(* IEC 61131-3 sources: TIA2AX/tests/V18/test_projects/expected/HW_2200330/ST70_PLC, 7 files *)

(* ---- HwIdentifiers.st ---- *)
TYPE
	HwIdentifiers : WORD
	(
		ST70_PLC_Profilschiene_0 :=	WORD#256,
		ST70_PLC :=	WORD#48,
		ST70_PLC_Card_reader_writer_1 :=	WORD#51,
		ST70_PLC_CPU_display_1 :=	WORD#54,
		ST70_PLC_OPC_UA_1 :=	WORD#117,
		ST70_PLC_DP_interface_1 :=	WORD#60,
		ST70_PLC_PROFINET_interface_1 :=	WORD#64,
		ST70_PLC_PROFINET_interface_1_Port_1 :=	WORD#65,
		ST70_PLC_PROFINET_interface_1_Port_2 :=	WORD#66,
		ST70_PLC_PROFINET_interface_2 :=	WORD#72,
		ST70_PLC_PROFINET_interface_2_Port_1 :=	WORD#73,
		ST70_Switch_SCALANCE_X_rack :=	WORD#406,
		ST70_Switch :=	WORD#407,
		ST70_Switch_ST70_Switch :=	WORD#408,
		ST70_Switch_SCALANCE_interface_1 :=	WORD#409,
		ST70_Switch_SCALANCE_interface_1_Port_1 :=	WORD#410,
		ST70_Switch_SCALANCE_interface_1_Port_2 :=	WORD#411,
		ST70_Switch_SCALANCE_interface_1_Port_3 :=	WORD#412,
		ST70_Switch_SCALANCE_interface_1_Port_4 :=	WORD#413,
		ST70_Switch_SCALANCE_interface_1_Port_5 :=	WORD#414,
		ST70_Switch_SCALANCE_interface_1_Port_6 :=	WORD#415,
		ST70_Switch_SCALANCE_interface_1_Port_7 :=	WORD#416,
		ST70_Switch_SCALANCE_interface_1_Port_8 :=	WORD#417,
		ST70_Switch_SCALANCE_interface_1_Port_9 :=	WORD#418,
		ST70_Switch_SCALANCE_interface_1_Port_10 :=	WORD#419,
		ST70_Switch_SCALANCE_interface_1_Port_11 :=	WORD#420,
		ST70_Switch_SCALANCE_interface_1_Port_12 :=	WORD#421,
		ST70_Switch_SCALANCE_interface_1_Port_13 :=	WORD#422,
		ST70_Switch_SCALANCE_interface_1_Port_14 :=	WORD#423,
		ST70_Switch_SCALANCE_interface_1_Port_15 :=	WORD#424,
		ST70_Switch_SCALANCE_interface_1_Port_16 :=	WORD#425,
		ST70_HMI_ConnectionBox_Connection_Box :=	WORD#265,
		ST70_HMI_ConnectionBox :=	WORD#258,
		ST70_HMI_ConnectionBox_ST70_HMI_ConnectionBox :=	WORD#259,
		ST70_HMI_ConnectionBox_SCALANCE_interface_1 :=	WORD#260,
		ST70_HMI_ConnectionBox_SCALANCE_interface_1_Port_1 :=	WORD#261,
		ST70_HMI_ConnectionBox_SCALANCE_interface_1_Port_2 :=	WORD#262,
		ST70_HMI_ConnectionBox_SCALANCE_interface_1_Port_3 :=	WORD#263,
		ST70_ET200SP_Rack_0 :=	WORD#272,
		ST70_ET200SP :=	WORD#273,
		ST70_ET200SP_ST70_ET200SP :=	WORD#274,
		ST70_ET200SP_PROFINET_interface :=	WORD#275,
		ST70_ET200SP_PROFINET_interface_Port_1 :=	WORD#277,
		ST70_ET200SP_PROFINET_interface_Port_2 :=	WORD#276,
		ST70_ET200SP_BA_2xRJ45 :=	WORD#277,
		ST70_ET200SP_CM_4xIO_Link_1 :=	WORD#278,
		ST70_ET200SP_DI_16x24VDC_ST_1 :=	WORD#279,
		ST70_ET200SP_DI_16x24VDC_ST_2 :=	WORD#280,
		ST70_ET200SP_DI_8x24VDC_ST_3 :=	WORD#281,
		ST70_ET200SP_DI_16x24VDC_ST_4 :=	WORD#266,
		ST70_ET200SP_DQ_16x24VDC_0_5A_ST_1 :=	WORD#267,
		ST70_ET200SP_DQ_16x24VDC_0_5A_ST_2 :=	WORD#268,
		ST70_ET200SP_DQ_16x24VDC_0_5A_ST_3 :=	WORD#269,
		ST70_ET200SP_Servermodul_1 :=	WORD#270,
		ST70_CPX_PN_IO_Interface :=	WORD#285,
		ST70_CPX_PN_IO_Interface_Port_1 :=	WORD#286,
		ST70_CPX_PN_IO_Interface_Port_2 :=	WORD#287,
		ST70_CPX_CPX :=	WORD#288,
		ST70_CPX_MPA1S_VMPA1_FB_EMS_8_8DO_1 :=	WORD#289,
		ST70_CPX_MPA1S_VMPA1_FB_EMS_8_8DO_2 :=	WORD#290,
		ST70_CPX_MPA1S_VMPA1_FB_EMS_8_8DO_3 :=	WORD#291,
		ST70_CPX_MPA2S_VMPA2_FB_EMS_4_4DO_1 :=	WORD#292,
		ST70_CPX_MPA1G_VMPA1_FB_EMG_8_8DO_3 :=	WORD#293,
		ST70_1_DM260_PB_Rack :=	WORD#295,
		ST70_1_DM260_PB :=	WORD#296,
		ST70_1_DM260_PB_Interface :=	WORD#297,
		ST70_1_DM260_PB_Interface_Port_1 :=	WORD#298,
		ST70_1_DM260_PB_DataMan_260 :=	WORD#299,
		ST70_1_DM260_PB_Acquisition_Control_1 :=	WORD#300,
		ST70_1_DM260_PB_Acquisition_Status_1 :=	WORD#301,
		ST70_1_DM260_PB_Results_Control_1 :=	WORD#302,
		ST70_1_DM260_PB_Results_Status_1 :=	WORD#303,
		ST70_1_DM260_PB_Soft_Event_Control_1 :=	WORD#304,
		ST70_1_DM260_PB_User_Data_64_bytes_1 :=	WORD#305,
		ST70_1_DM260_PB_Result_Data_64_bytes_1 :=	WORD#306,
		ST70_2_DM260_PB_Rack :=	WORD#308,
		ST70_2_DM260_PB :=	WORD#309,
		ST70_2_DM260_PB_Interface :=	WORD#310,
		ST70_2_DM260_PB_Interface_Port_1 :=	WORD#311,
		ST70_2_DM260_PB_DataMan_260 :=	WORD#312,
		ST70_2_DM260_PB_Acquisition_Control_1 :=	WORD#313,
		ST70_2_DM260_PB_Acquisition_Status_1 :=	WORD#314,
		ST70_2_DM260_PB_Results_Control_1 :=	WORD#315,
		ST70_2_DM260_PB_Results_Status_1 :=	WORD#316,
		ST70_2_DM260_PB_Soft_Event_Control_1 :=	WORD#317,
		ST70_2_DM260_PB_User_Data_64_bytes_1 :=	WORD#318,
		ST70_2_DM260_PB_Result_Data_64_bytes_1 :=	WORD#319,
		ST70_1_CMMT_3GF1_PN_IO_Interface :=	WORD#323,
		ST70_1_CMMT_3GF1_PN_IO_Interface_Port_1 :=	WORD#324,
		ST70_1_CMMT_3GF1_PN_IO_Interface_Port_2 :=	WORD#325,
		ST70_1_CMMT_3GF1_CMMT_AS_V1 :=	WORD#326,
		ST70_1_CMMT_3GF1_DO_SERVO_1_Module_Access_Point :=	WORD#328,
		ST70_1_CMMT_3GF1_DO_SERVO_1_Siemens_telegram_111_PZD_12_12 :=	WORD#329,
		ST70_1_CMMT_3GF1_Siemens_telegram_111_PZD_12_12 :=	WORD#329,
		ST70_1_CMMT_3GF2_PN_IO_Interface :=	WORD#333,
		ST70_1_CMMT_3GF2_PN_IO_Interface_Port_1 :=	WORD#334,
		ST70_1_CMMT_3GF2_PN_IO_Interface_Port_2 :=	WORD#335,
		ST70_1_CMMT_3GF2_CMMT_AS_V1 :=	WORD#336,
		ST70_1_CMMT_3GF2_DO_SERVO_1_Module_Access_Point :=	WORD#338,
		ST70_1_CMMT_3GF2_DO_SERVO_1_Siemens_telegram_111_PZD_12_12 :=	WORD#339,
		ST70_1_CMMT_3GF2_Siemens_telegram_111_PZD_12_12 :=	WORD#339,
		ST70_3_DM260_PB_Rack :=	WORD#341,
		ST70_3_DM260_PB :=	WORD#342,
		ST70_3_DM260_PB_Interface :=	WORD#343,
		ST70_3_DM260_PB_Interface_Port_1 :=	WORD#344,
		ST70_3_DM260_PB_DataMan_260 :=	WORD#345,
		ST70_3_DM260_PB_Acquisition_Control_1 :=	WORD#346,
		ST70_3_DM260_PB_Acquisition_Status_1 :=	WORD#347,
		ST70_3_DM260_PB_Results_Control_1 :=	WORD#348,
		ST70_3_DM260_PB_Results_Status_1 :=	WORD#349,
		ST70_3_DM260_PB_Soft_Event_Control_1 :=	WORD#350,
		ST70_3_DM260_PB_User_Data_64_bytes_1 :=	WORD#351,
		ST70_3_DM260_PB_Result_Data_64_bytes_1 :=	WORD#352,
		ST70_1_DM260_EB_Rack :=	WORD#354,
		ST70_1_DM260_EB :=	WORD#355,
		ST70_1_DM260_EB_Interface :=	WORD#356,
		ST70_1_DM260_EB_Interface_Port_1 :=	WORD#357,
		ST70_1_DM260_EB_DataMan_260 :=	WORD#358,
		ST70_1_DM260_EB_Acquisition_Control_1 :=	WORD#359,
		ST70_1_DM260_EB_Acquisition_Status_1 :=	WORD#360,
		ST70_1_DM260_EB_Results_Control_1 :=	WORD#361,
		ST70_1_DM260_EB_Results_Status_1 :=	WORD#362,
		ST70_1_DM260_EB_Soft_Event_Control_1 :=	WORD#363,
		ST70_1_DM260_EB_User_Data_64_bytes_1 :=	WORD#364,
		ST70_1_DM260_EB_Result_Data_64_bytes_1 :=	WORD#365,
		ST70_2_DM260_EB_Rack :=	WORD#367,
		ST70_2_DM260_EB :=	WORD#368,
		ST70_2_DM260_EB_Interface :=	WORD#369,
		ST70_2_DM260_EB_Interface_Port_1 :=	WORD#370,
		ST70_2_DM260_EB_DataMan_260 :=	WORD#371,
		ST70_2_DM260_EB_Acquisition_Control_1 :=	WORD#372,
		ST70_2_DM260_EB_Acquisition_Status_1 :=	WORD#373,
		ST70_2_DM260_EB_Results_Control_1 :=	WORD#374,
		ST70_2_DM260_EB_Results_Status_1 :=	WORD#375,
		ST70_2_DM260_EB_Soft_Event_Control_1 :=	WORD#376,
		ST70_2_DM260_EB_User_Data_64_bytes_1 :=	WORD#377,
		ST70_2_DM260_EB_Result_Data_64_bytes_1 :=	WORD#378,
		ST70_3_DM260_EB_Rack :=	WORD#380,
		ST70_3_DM260_EB :=	WORD#381,
		ST70_3_DM260_EB_Interface :=	WORD#382,
		ST70_3_DM260_EB_Interface_Port_1 :=	WORD#383,
		ST70_3_DM260_EB_DataMan_260 :=	WORD#384,
		ST70_3_DM260_EB_Acquisition_Control_1 :=	WORD#385,
		ST70_3_DM260_EB_Acquisition_Status_1 :=	WORD#386,
		ST70_3_DM260_EB_Results_Control_1 :=	WORD#387,
		ST70_3_DM260_EB_Results_Status_1 :=	WORD#388,
		ST70_3_DM260_EB_Soft_Event_Control_1 :=	WORD#389,
		ST70_3_DM260_EB_User_Data_64_bytes_1 :=	WORD#390,
		ST70_3_DM260_EB_Result_Data_64_bytes_1 :=	WORD#391,
		ST70_1_CMMT_3GF3_PN_IO_Interface :=	WORD#395,
		ST70_1_CMMT_3GF3_PN_IO_Interface_Port_1 :=	WORD#396,
		ST70_1_CMMT_3GF3_PN_IO_Interface_Port_2 :=	WORD#397,
		ST70_1_CMMT_3GF3_CMMT_AS_V1 :=	WORD#398,
		ST70_1_CMMT_3GF3_DO_SERVO_1_Module_Access_Point :=	WORD#400,
		ST70_1_CMMT_3GF3_DO_SERVO_1_Siemens_telegram_111_PZD_12_12 :=	WORD#401,
		ST70_1_CMMT_3GF3_Siemens_telegram_111_PZD_12_12 :=	WORD#401,
		NONE:= WORD#0
	);
END_TYPE

(* ---- HwInputs.st ---- *)
TYPE
	HwInputs : STRUCT
		ST70_ET200SP_CM_4xIO_Link_1 AT %B100 : ARRAY[0..31] OF BYTE;
		ST70_ET200SP_DI_16x24VDC_ST_1 AT %B0 : WORD;
		ST70_ET200SP_DI_16x24VDC_ST_2 AT %B2 : WORD;
		ST70_ET200SP_DI_8x24VDC_ST_3 AT %B4 : BYTE;
		ST70_ET200SP_DI_16x24VDC_ST_4 AT %B5 : WORD;
		ST70_1_DM260_PB_Acquisition_Status_1 AT %B1000 : ARRAY[0..2] OF BYTE;
		ST70_1_DM260_PB_Results_Status_1 AT %B1003 : BYTE;
		ST70_1_DM260_PB_Soft_Event_Control_1 AT %B1004 : BYTE;
		ST70_1_DM260_PB_Result_Data_64_bytes_1 AT %B1010 : ARRAY[0..71] OF BYTE;
		ST70_2_DM260_PB_Acquisition_Status_1 AT %B2000 : ARRAY[0..2] OF BYTE;
		ST70_2_DM260_PB_Results_Status_1 AT %B2003 : BYTE;
		ST70_2_DM260_PB_Soft_Event_Control_1 AT %B2004 : BYTE;
		ST70_2_DM260_PB_Result_Data_64_bytes_1 AT %B2010 : ARRAY[0..71] OF BYTE;
		ST70_1_CMMT_3GF1_DO_SERVO_1_Siemens_telegram_111_PZD_12_12 AT %B1500 : ARRAY[0..23] OF BYTE;
		ST70_1_CMMT_3GF2_DO_SERVO_1_Siemens_telegram_111_PZD_12_12 AT %B1600 : ARRAY[0..23] OF BYTE;
		ST70_3_DM260_PB_Acquisition_Status_1 AT %B3000 : ARRAY[0..2] OF BYTE;
		ST70_3_DM260_PB_Results_Status_1 AT %B3003 : BYTE;
		ST70_3_DM260_PB_Soft_Event_Control_1 AT %B3004 : BYTE;
		ST70_3_DM260_PB_Result_Data_64_bytes_1 AT %B3010 : ARRAY[0..71] OF BYTE;
		ST70_1_DM260_EB_Acquisition_Status_1 AT %B1200 : ARRAY[0..2] OF BYTE;
		ST70_1_DM260_EB_Results_Status_1 AT %B1203 : BYTE;
		ST70_1_DM260_EB_Soft_Event_Control_1 AT %B1204 : BYTE;
		ST70_1_DM260_EB_Result_Data_64_bytes_1 AT %B1210 : ARRAY[0..71] OF BYTE;
		ST70_2_DM260_EB_Acquisition_Status_1 AT %B2200 : ARRAY[0..2] OF BYTE;
		ST70_2_DM260_EB_Results_Status_1 AT %B2203 : BYTE;
		ST70_2_DM260_EB_Soft_Event_Control_1 AT %B2204 : BYTE;
		ST70_2_DM260_EB_Result_Data_64_bytes_1 AT %B2210 : ARRAY[0..71] OF BYTE;
		ST70_3_DM260_EB_Acquisition_Status_1 AT %B3200 : ARRAY[0..2] OF BYTE;
		ST70_3_DM260_EB_Results_Status_1 AT %B3203 : BYTE;
		ST70_3_DM260_EB_Soft_Event_Control_1 AT %B3204 : BYTE;
		ST70_3_DM260_EB_Result_Data_64_bytes_1 AT %B3210 : ARRAY[0..71] OF BYTE;
		ST70_1_CMMT_3GF3_DO_SERVO_1_Siemens_telegram_111_PZD_12_12 AT %B1624 : ARRAY[0..23] OF BYTE;
	END_STRUCT;
END_TYPE

(* ---- HwOutputs.st ---- *)
TYPE
	HwOutputs : STRUCT
		ST70_ET200SP_CM_4xIO_Link_1 AT %B100 : ARRAY[0..31] OF BYTE;
		ST70_ET200SP_DQ_16x24VDC_0_5A_ST_1 AT %B0 : WORD;
		ST70_ET200SP_DQ_16x24VDC_0_5A_ST_2 AT %B2 : WORD;
		ST70_ET200SP_DQ_16x24VDC_0_5A_ST_3 AT %B4 : WORD;
		ST70_CPX_MPA1S_VMPA1_FB_EMS_8_8DO_1 AT %B200 : BYTE;
		ST70_CPX_MPA1S_VMPA1_FB_EMS_8_8DO_2 AT %B201 : BYTE;
		ST70_CPX_MPA1S_VMPA1_FB_EMS_8_8DO_3 AT %B202 : BYTE;
		ST70_CPX_MPA2S_VMPA2_FB_EMS_4_4DO_1 AT %B6 : BYTE;
		ST70_CPX_MPA1G_VMPA1_FB_EMG_8_8DO_3 AT %B204 : BYTE;
		ST70_1_DM260_PB_Acquisition_Control_1 AT %B1000 : BYTE;
		ST70_1_DM260_PB_Results_Control_1 AT %B1003 : BYTE;
		ST70_1_DM260_PB_Soft_Event_Control_1 AT %B1004 : BYTE;
		ST70_1_DM260_PB_User_Data_64_bytes_1 AT %B1010 : ARRAY[0..67] OF BYTE;
		ST70_2_DM260_PB_Acquisition_Control_1 AT %B2000 : BYTE;
		ST70_2_DM260_PB_Results_Control_1 AT %B2003 : BYTE;
		ST70_2_DM260_PB_Soft_Event_Control_1 AT %B2004 : BYTE;
		ST70_2_DM260_PB_User_Data_64_bytes_1 AT %B2010 : ARRAY[0..67] OF BYTE;
		ST70_1_CMMT_3GF1_DO_SERVO_1_Siemens_telegram_111_PZD_12_12 AT %B1500 : ARRAY[0..23] OF BYTE;
		ST70_1_CMMT_3GF2_DO_SERVO_1_Siemens_telegram_111_PZD_12_12 AT %B1600 : ARRAY[0..23] OF BYTE;
		ST70_3_DM260_PB_Acquisition_Control_1 AT %B3000 : BYTE;
		ST70_3_DM260_PB_Results_Control_1 AT %B3003 : BYTE;
		ST70_3_DM260_PB_Soft_Event_Control_1 AT %B3004 : BYTE;
		ST70_3_DM260_PB_User_Data_64_bytes_1 AT %B3010 : ARRAY[0..67] OF BYTE;
		ST70_1_DM260_EB_Acquisition_Control_1 AT %B1200 : BYTE;
		ST70_1_DM260_EB_Results_Control_1 AT %B1203 : BYTE;
		ST70_1_DM260_EB_Soft_Event_Control_1 AT %B1204 : BYTE;
		ST70_1_DM260_EB_User_Data_64_bytes_1 AT %B1210 : ARRAY[0..67] OF BYTE;
		ST70_2_DM260_EB_Acquisition_Control_1 AT %B2200 : BYTE;
		ST70_2_DM260_EB_Results_Control_1 AT %B2203 : BYTE;
		ST70_2_DM260_EB_Soft_Event_Control_1 AT %B2204 : BYTE;
		ST70_2_DM260_EB_User_Data_64_bytes_1 AT %B2210 : ARRAY[0..67] OF BYTE;
		ST70_3_DM260_EB_Acquisition_Control_1 AT %B3200 : BYTE;
		ST70_3_DM260_EB_Results_Control_1 AT %B3203 : BYTE;
		ST70_3_DM260_EB_Soft_Event_Control_1 AT %B3204 : BYTE;
		ST70_3_DM260_EB_User_Data_64_bytes_1 AT %B3210 : ARRAY[0..67] OF BYTE;
		ST70_1_CMMT_3GF3_DO_SERVO_1_Siemens_telegram_111_PZD_12_12 AT %B1624 : ARRAY[0..23] OF BYTE;
	END_STRUCT;
END_TYPE

(* ---- PlcInputs.st ---- *)
TYPE
	PlcInputs : STRUCT
		ST70_ET200SP_CM_4xIO_Link_1 : ARRAY[0..31] OF BYTE;
		ST70_ET200SP_DI_16x24VDC_ST_1 : WORD;
		ST70_ET200SP_DI_16x24VDC_ST_2 : WORD;
		ST70_ET200SP_DI_8x24VDC_ST_3 : BYTE;
		ST70_ET200SP_DI_16x24VDC_ST_4 : WORD;
		ST70_1_DM260_PB_Acquisition_Status_1 : ARRAY[0..2] OF BYTE;
		ST70_1_DM260_PB_Results_Status_1 : BYTE;
		ST70_1_DM260_PB_Soft_Event_Control_1 : BYTE;
		ST70_1_DM260_PB_Result_Data_64_bytes_1 : ARRAY[0..71] OF BYTE;
		ST70_2_DM260_PB_Acquisition_Status_1 : ARRAY[0..2] OF BYTE;
		ST70_2_DM260_PB_Results_Status_1 : BYTE;
		ST70_2_DM260_PB_Soft_Event_Control_1 : BYTE;
		ST70_2_DM260_PB_Result_Data_64_bytes_1 : ARRAY[0..71] OF BYTE;
		ST70_1_CMMT_3GF1_DO_SERVO_1_Siemens_telegram_111_PZD_12_12 : ARRAY[0..23] OF BYTE;
		ST70_1_CMMT_3GF2_DO_SERVO_1_Siemens_telegram_111_PZD_12_12 : ARRAY[0..23] OF BYTE;
		ST70_3_DM260_PB_Acquisition_Status_1 : ARRAY[0..2] OF BYTE;
		ST70_3_DM260_PB_Results_Status_1 : BYTE;
		ST70_3_DM260_PB_Soft_Event_Control_1 : BYTE;
		ST70_3_DM260_PB_Result_Data_64_bytes_1 : ARRAY[0..71] OF BYTE;
		ST70_1_DM260_EB_Acquisition_Status_1 : ARRAY[0..2] OF BYTE;
		ST70_1_DM260_EB_Results_Status_1 : BYTE;
		ST70_1_DM260_EB_Soft_Event_Control_1 : BYTE;
		ST70_1_DM260_EB_Result_Data_64_bytes_1 : ARRAY[0..71] OF BYTE;
		ST70_2_DM260_EB_Acquisition_Status_1 : ARRAY[0..2] OF BYTE;
		ST70_2_DM260_EB_Results_Status_1 : BYTE;
		ST70_2_DM260_EB_Soft_Event_Control_1 : BYTE;
		ST70_2_DM260_EB_Result_Data_64_bytes_1 : ARRAY[0..71] OF BYTE;
		ST70_3_DM260_EB_Acquisition_Status_1 : ARRAY[0..2] OF BYTE;
		ST70_3_DM260_EB_Results_Status_1 : BYTE;
		ST70_3_DM260_EB_Soft_Event_Control_1 : BYTE;
		ST70_3_DM260_EB_Result_Data_64_bytes_1 : ARRAY[0..71] OF BYTE;
		ST70_1_CMMT_3GF3_DO_SERVO_1_Siemens_telegram_111_PZD_12_12 : ARRAY[0..23] OF BYTE;
	END_STRUCT;
END_TYPE

(* ---- PlcOutputs.st ---- *)
TYPE
	PlcOutputs : STRUCT
		ST70_ET200SP_CM_4xIO_Link_1 : ARRAY[0..31] OF BYTE;
		ST70_ET200SP_DQ_16x24VDC_0_5A_ST_1 : WORD;
		ST70_ET200SP_DQ_16x24VDC_0_5A_ST_2 : WORD;
		ST70_ET200SP_DQ_16x24VDC_0_5A_ST_3 : WORD;
		ST70_CPX_MPA1S_VMPA1_FB_EMS_8_8DO_1 : BYTE;
		ST70_CPX_MPA1S_VMPA1_FB_EMS_8_8DO_2 : BYTE;
		ST70_CPX_MPA1S_VMPA1_FB_EMS_8_8DO_3 : BYTE;
		ST70_CPX_MPA2S_VMPA2_FB_EMS_4_4DO_1 : BYTE;
		ST70_CPX_MPA1G_VMPA1_FB_EMG_8_8DO_3 : BYTE;
		ST70_1_DM260_PB_Acquisition_Control_1 : BYTE;
		ST70_1_DM260_PB_Results_Control_1 : BYTE;
		ST70_1_DM260_PB_Soft_Event_Control_1 : BYTE;
		ST70_1_DM260_PB_User_Data_64_bytes_1 : ARRAY[0..67] OF BYTE;
		ST70_2_DM260_PB_Acquisition_Control_1 : BYTE;
		ST70_2_DM260_PB_Results_Control_1 : BYTE;
		ST70_2_DM260_PB_Soft_Event_Control_1 : BYTE;
		ST70_2_DM260_PB_User_Data_64_bytes_1 : ARRAY[0..67] OF BYTE;
		ST70_1_CMMT_3GF1_DO_SERVO_1_Siemens_telegram_111_PZD_12_12 : ARRAY[0..23] OF BYTE;
		ST70_1_CMMT_3GF2_DO_SERVO_1_Siemens_telegram_111_PZD_12_12 : ARRAY[0..23] OF BYTE;
		ST70_3_DM260_PB_Acquisition_Control_1 : BYTE;
		ST70_3_DM260_PB_Results_Control_1 : BYTE;
		ST70_3_DM260_PB_Soft_Event_Control_1 : BYTE;
		ST70_3_DM260_PB_User_Data_64_bytes_1 : ARRAY[0..67] OF BYTE;
		ST70_1_DM260_EB_Acquisition_Control_1 : BYTE;
		ST70_1_DM260_EB_Results_Control_1 : BYTE;
		ST70_1_DM260_EB_Soft_Event_Control_1 : BYTE;
		ST70_1_DM260_EB_User_Data_64_bytes_1 : ARRAY[0..67] OF BYTE;
		ST70_2_DM260_EB_Acquisition_Control_1 : BYTE;
		ST70_2_DM260_EB_Results_Control_1 : BYTE;
		ST70_2_DM260_EB_Soft_Event_Control_1 : BYTE;
		ST70_2_DM260_EB_User_Data_64_bytes_1 : ARRAY[0..67] OF BYTE;
		ST70_3_DM260_EB_Acquisition_Control_1 : BYTE;
		ST70_3_DM260_EB_Results_Control_1 : BYTE;
		ST70_3_DM260_EB_Soft_Event_Control_1 : BYTE;
		ST70_3_DM260_EB_User_Data_64_bytes_1 : ARRAY[0..67] OF BYTE;
		ST70_1_CMMT_3GF3_DO_SERVO_1_Siemens_telegram_111_PZD_12_12 : ARRAY[0..23] OF BYTE;
	END_STRUCT;
END_TYPE

(* ---- CopyInputs.st ---- *)
FUNCTION CopyInputs
	VAR_EXTERNAL
		HwInputs : HwInputs;
		PlcInputs : PlcInputs;
	END_VAR
	PlcInputs.ST70_ET200SP_CM_4xIO_Link_1[0] := HwInputs.ST70_ET200SP_CM_4xIO_Link_1[0];
	PlcInputs.ST70_ET200SP_CM_4xIO_Link_1[1] := HwInputs.ST70_ET200SP_CM_4xIO_Link_1[1];
	PlcInputs.ST70_ET200SP_CM_4xIO_Link_1[2] := HwInputs.ST70_ET200SP_CM_4xIO_Link_1[2];
	PlcInputs.ST70_ET200SP_CM_4xIO_Link_1[3] := HwInputs.ST70_ET200SP_CM_4xIO_Link_1[3];
	PlcInputs.ST70_ET200SP_CM_4xIO_Link_1[4] := HwInputs.ST70_ET200SP_CM_4xIO_Link_1[4];
	PlcInputs.ST70_ET200SP_CM_4xIO_Link_1[5] := HwInputs.ST70_ET200SP_CM_4xIO_Link_1[5];
	PlcInputs.ST70_ET200SP_CM_4xIO_Link_1[6] := HwInputs.ST70_ET200SP_CM_4xIO_Link_1[6];
	PlcInputs.ST70_ET200SP_CM_4xIO_Link_1[7] := HwInputs.ST70_ET200SP_CM_4xIO_Link_1[7];
	PlcInputs.ST70_ET200SP_CM_4xIO_Link_1[8] := HwInputs.ST70_ET200SP_CM_4xIO_Link_1[8];
	PlcInputs.ST70_ET200SP_CM_4xIO_Link_1[9] := HwInputs.ST70_ET200SP_CM_4xIO_Link_1[9];
	PlcInputs.ST70_ET200SP_CM_4xIO_Link_1[10] := HwInputs.ST70_ET200SP_CM_4xIO_Link_1[10];
	PlcInputs.ST70_ET200SP_CM_4xIO_Link_1[11] := HwInputs.ST70_ET200SP_CM_4xIO_Link_1[11];
	PlcInputs.ST70_ET200SP_CM_4xIO_Link_1[12] := HwInputs.ST70_ET200SP_CM_4xIO_Link_1[12];
	PlcInputs.ST70_ET200SP_CM_4xIO_Link_1[13] := HwInputs.ST70_ET200SP_CM_4xIO_Link_1[13];
	PlcInputs.ST70_ET200SP_CM_4xIO_Link_1[14] := HwInputs.ST70_ET200SP_CM_4xIO_Link_1[14];
	PlcInputs.ST70_ET200SP_CM_4xIO_Link_1[15] := HwInputs.ST70_ET200SP_CM_4xIO_Link_1[15];
	PlcInputs.ST70_ET200SP_CM_4xIO_Link_1[16] := HwInputs.ST70_ET200SP_CM_4xIO_Link_1[16];
	PlcInputs.ST70_ET200SP_CM_4xIO_Link_1[17] := HwInputs.ST70_ET200SP_CM_4xIO_Link_1[17];
	PlcInputs.ST70_ET200SP_CM_4xIO_Link_1[18] := HwInputs.ST70_ET200SP_CM_4xIO_Link_1[18];
	PlcInputs.ST70_ET200SP_CM_4xIO_Link_1[19] := HwInputs.ST70_ET200SP_CM_4xIO_Link_1[19];
	PlcInputs.ST70_ET200SP_CM_4xIO_Link_1[20] := HwInputs.ST70_ET200SP_CM_4xIO_Link_1[20];
	PlcInputs.ST70_ET200SP_CM_4xIO_Link_1[21] := HwInputs.ST70_ET200SP_CM_4xIO_Link_1[21];
	PlcInputs.ST70_ET200SP_CM_4xIO_Link_1[22] := HwInputs.ST70_ET200SP_CM_4xIO_Link_1[22];
	PlcInputs.ST70_ET200SP_CM_4xIO_Link_1[23] := HwInputs.ST70_ET200SP_CM_4xIO_Link_1[23];
	PlcInputs.ST70_ET200SP_CM_4xIO_Link_1[24] := HwInputs.ST70_ET200SP_CM_4xIO_Link_1[24];
	PlcInputs.ST70_ET200SP_CM_4xIO_Link_1[25] := HwInputs.ST70_ET200SP_CM_4xIO_Link_1[25];
	PlcInputs.ST70_ET200SP_CM_4xIO_Link_1[26] := HwInputs.ST70_ET200SP_CM_4xIO_Link_1[26];
	PlcInputs.ST70_ET200SP_CM_4xIO_Link_1[27] := HwInputs.ST70_ET200SP_CM_4xIO_Link_1[27];
	PlcInputs.ST70_ET200SP_CM_4xIO_Link_1[28] := HwInputs.ST70_ET200SP_CM_4xIO_Link_1[28];
	PlcInputs.ST70_ET200SP_CM_4xIO_Link_1[29] := HwInputs.ST70_ET200SP_CM_4xIO_Link_1[29];
	PlcInputs.ST70_ET200SP_CM_4xIO_Link_1[30] := HwInputs.ST70_ET200SP_CM_4xIO_Link_1[30];
	PlcInputs.ST70_ET200SP_CM_4xIO_Link_1[31] := HwInputs.ST70_ET200SP_CM_4xIO_Link_1[31];
	PlcInputs.ST70_ET200SP_DI_16x24VDC_ST_1 := HwInputs.ST70_ET200SP_DI_16x24VDC_ST_1;
	PlcInputs.ST70_ET200SP_DI_16x24VDC_ST_2 := HwInputs.ST70_ET200SP_DI_16x24VDC_ST_2;
	PlcInputs.ST70_ET200SP_DI_8x24VDC_ST_3 := HwInputs.ST70_ET200SP_DI_8x24VDC_ST_3;
	PlcInputs.ST70_ET200SP_DI_16x24VDC_ST_4 := HwInputs.ST70_ET200SP_DI_16x24VDC_ST_4;
	PlcInputs.ST70_1_DM260_PB_Acquisition_Status_1[0] := HwInputs.ST70_1_DM260_PB_Acquisition_Status_1[0];
	PlcInputs.ST70_1_DM260_PB_Acquisition_Status_1[1] := HwInputs.ST70_1_DM260_PB_Acquisition_Status_1[1];
	PlcInputs.ST70_1_DM260_PB_Acquisition_Status_1[2] := HwInputs.ST70_1_DM260_PB_Acquisition_Status_1[2];
	PlcInputs.ST70_1_DM260_PB_Results_Status_1 := HwInputs.ST70_1_DM260_PB_Results_Status_1;
	PlcInputs.ST70_1_DM260_PB_Soft_Event_Control_1 := HwInputs.ST70_1_DM260_PB_Soft_Event_Control_1;
	PlcInputs.ST70_1_DM260_PB_Result_Data_64_bytes_1[0] := HwInputs.ST70_1_DM260_PB_Result_Data_64_bytes_1[0];
	PlcInputs.ST70_1_DM260_PB_Result_Data_64_bytes_1[1] := HwInputs.ST70_1_DM260_PB_Result_Data_64_bytes_1[1];
	PlcInputs.ST70_1_DM260_PB_Result_Data_64_bytes_1[2] := HwInputs.ST70_1_DM260_PB_Result_Data_64_bytes_1[2];
	PlcInputs.ST70_1_DM260_PB_Result_Data_64_bytes_1[3] := HwInputs.ST70_1_DM260_PB_Result_Data_64_bytes_1[3];
	PlcInputs.ST70_1_DM260_PB_Result_Data_64_bytes_1[4] := HwInputs.ST70_1_DM260_PB_Result_Data_64_bytes_1[4];
	PlcInputs.ST70_1_DM260_PB_Result_Data_64_bytes_1[5] := HwInputs.ST70_1_DM260_PB_Result_Data_64_bytes_1[5];
	PlcInputs.ST70_1_DM260_PB_Result_Data_64_bytes_1[6] := HwInputs.ST70_1_DM260_PB_Result_Data_64_bytes_1[6];
	PlcInputs.ST70_1_DM260_PB_Result_Data_64_bytes_1[7] := HwInputs.ST70_1_DM260_PB_Result_Data_64_bytes_1[7];
	PlcInputs.ST70_1_DM260_PB_Result_Data_64_bytes_1[8] := HwInputs.ST70_1_DM260_PB_Result_Data_64_bytes_1[8];
	PlcInputs.ST70_1_DM260_PB_Result_Data_64_bytes_1[9] := HwInputs.ST70_1_DM260_PB_Result_Data_64_bytes_1[9];
	PlcInputs.ST70_1_DM260_PB_Result_Data_64_bytes_1[10] := HwInputs.ST70_1_DM260_PB_Result_Data_64_bytes_1[10];
	PlcInputs.ST70_1_DM260_PB_Result_Data_64_bytes_1[11] := HwInputs.ST70_1_DM260_PB_Result_Data_64_bytes_1[11];
	PlcInputs.ST70_1_DM260_PB_Result_Data_64_bytes_1[12] := HwInputs.ST70_1_DM260_PB_Result_Data_64_bytes_1[12];
	PlcInputs.ST70_1_DM260_PB_Result_Data_64_bytes_1[13] := HwInputs.ST70_1_DM260_PB_Result_Data_64_bytes_1[13];
	PlcInputs.ST70_1_DM260_PB_Result_Data_64_bytes_1[14] := HwInputs.ST70_1_DM260_PB_Result_Data_64_bytes_1[14];
	PlcInputs.ST70_1_DM260_PB_Result_Data_64_bytes_1[15] := HwInputs.ST70_1_DM260_PB_Result_Data_64_bytes_1[15];
	PlcInputs.ST70_1_DM260_PB_Result_Data_64_bytes_1[16] := HwInputs.ST70_1_DM260_PB_Result_Data_64_bytes_1[16];
	PlcInputs.ST70_1_DM260_PB_Result_Data_64_bytes_1[17] := HwInputs.ST70_1_DM260_PB_Result_Data_64_bytes_1[17];
	PlcInputs.ST70_1_DM260_PB_Result_Data_64_bytes_1[18] := HwInputs.ST70_1_DM260_PB_Result_Data_64_bytes_1[18];
	PlcInputs.ST70_1_DM260_PB_Result_Data_64_bytes_1[19] := HwInputs.ST70_1_DM260_PB_Result_Data_64_bytes_1[19];
	PlcInputs.ST70_1_DM260_PB_Result_Data_64_bytes_1[20] := HwInputs.ST70_1_DM260_PB_Result_Data_64_bytes_1[20];
	PlcInputs.ST70_1_DM260_PB_Result_Data_64_bytes_1[21] := HwInputs.ST70_1_DM260_PB_Result_Data_64_bytes_1[21];
	PlcInputs.ST70_1_DM260_PB_Result_Data_64_bytes_1[22] := HwInputs.ST70_1_DM260_PB_Result_Data_64_bytes_1[22];
	PlcInputs.ST70_1_DM260_PB_Result_Data_64_bytes_1[23] := HwInputs.ST70_1_DM260_PB_Result_Data_64_bytes_1[23];
	PlcInputs.ST70_1_DM260_PB_Result_Data_64_bytes_1[24] := HwInputs.ST70_1_DM260_PB_Result_Data_64_bytes_1[24];
	PlcInputs.ST70_1_DM260_PB_Result_Data_64_bytes_1[25] := HwInputs.ST70_1_DM260_PB_Result_Data_64_bytes_1[25];
	PlcInputs.ST70_1_DM260_PB_Result_Data_64_bytes_1[26] := HwInputs.ST70_1_DM260_PB_Result_Data_64_bytes_1[26];
	PlcInputs.ST70_1_DM260_PB_Result_Data_64_bytes_1[27] := HwInputs.ST70_1_DM260_PB_Result_Data_64_bytes_1[27];
	PlcInputs.ST70_1_DM260_PB_Result_Data_64_bytes_1[28] := HwInputs.ST70_1_DM260_PB_Result_Data_64_bytes_1[28];
	PlcInputs.ST70_1_DM260_PB_Result_Data_64_bytes_1[29] := HwInputs.ST70_1_DM260_PB_Result_Data_64_bytes_1[29];
	PlcInputs.ST70_1_DM260_PB_Result_Data_64_bytes_1[30] := HwInputs.ST70_1_DM260_PB_Result_Data_64_bytes_1[30];
	PlcInputs.ST70_1_DM260_PB_Result_Data_64_bytes_1[31] := HwInputs.ST70_1_DM260_PB_Result_Data_64_bytes_1[31];
	PlcInputs.ST70_1_DM260_PB_Result_Data_64_bytes_1[32] := HwInputs.ST70_1_DM260_PB_Result_Data_64_bytes_1[32];
	PlcInputs.ST70_1_DM260_PB_Result_Data_64_bytes_1[33] := HwInputs.ST70_1_DM260_PB_Result_Data_64_bytes_1[33];
	PlcInputs.ST70_1_DM260_PB_Result_Data_64_bytes_1[34] := HwInputs.ST70_1_DM260_PB_Result_Data_64_bytes_1[34];
	PlcInputs.ST70_1_DM260_PB_Result_Data_64_bytes_1[35] := HwInputs.ST70_1_DM260_PB_Result_Data_64_bytes_1[35];
	PlcInputs.ST70_1_DM260_PB_Result_Data_64_bytes_1[36] := HwInputs.ST70_1_DM260_PB_Result_Data_64_bytes_1[36];
	PlcInputs.ST70_1_DM260_PB_Result_Data_64_bytes_1[37] := HwInputs.ST70_1_DM260_PB_Result_Data_64_bytes_1[37];
	PlcInputs.ST70_1_DM260_PB_Result_Data_64_bytes_1[38] := HwInputs.ST70_1_DM260_PB_Result_Data_64_bytes_1[38];
	PlcInputs.ST70_1_DM260_PB_Result_Data_64_bytes_1[39] := HwInputs.ST70_1_DM260_PB_Result_Data_64_bytes_1[39];
	PlcInputs.ST70_1_DM260_PB_Result_Data_64_bytes_1[40] := HwInputs.ST70_1_DM260_PB_Result_Data_64_bytes_1[40];
	PlcInputs.ST70_1_DM260_PB_Result_Data_64_bytes_1[41] := HwInputs.ST70_1_DM260_PB_Result_Data_64_bytes_1[41];
	PlcInputs.ST70_1_DM260_PB_Result_Data_64_bytes_1[42] := HwInputs.ST70_1_DM260_PB_Result_Data_64_bytes_1[42];
	PlcInputs.ST70_1_DM260_PB_Result_Data_64_bytes_1[43] := HwInputs.ST70_1_DM260_PB_Result_Data_64_bytes_1[43];
	PlcInputs.ST70_1_DM260_PB_Result_Data_64_bytes_1[44] := HwInputs.ST70_1_DM260_PB_Result_Data_64_bytes_1[44];
	PlcInputs.ST70_1_DM260_PB_Result_Data_64_bytes_1[45] := HwInputs.ST70_1_DM260_PB_Result_Data_64_bytes_1[45];
	PlcInputs.ST70_1_DM260_PB_Result_Data_64_bytes_1[46] := HwInputs.ST70_1_DM260_PB_Result_Data_64_bytes_1[46];
	PlcInputs.ST70_1_DM260_PB_Result_Data_64_bytes_1[47] := HwInputs.ST70_1_DM260_PB_Result_Data_64_bytes_1[47];
	PlcInputs.ST70_1_DM260_PB_Result_Data_64_bytes_1[48] := HwInputs.ST70_1_DM260_PB_Result_Data_64_bytes_1[48];
	PlcInputs.ST70_1_DM260_PB_Result_Data_64_bytes_1[49] := HwInputs.ST70_1_DM260_PB_Result_Data_64_bytes_1[49];
	PlcInputs.ST70_1_DM260_PB_Result_Data_64_bytes_1[50] := HwInputs.ST70_1_DM260_PB_Result_Data_64_bytes_1[50];
	PlcInputs.ST70_1_DM260_PB_Result_Data_64_bytes_1[51] := HwInputs.ST70_1_DM260_PB_Result_Data_64_bytes_1[51];
	PlcInputs.ST70_1_DM260_PB_Result_Data_64_bytes_1[52] := HwInputs.ST70_1_DM260_PB_Result_Data_64_bytes_1[52];
	PlcInputs.ST70_1_DM260_PB_Result_Data_64_bytes_1[53] := HwInputs.ST70_1_DM260_PB_Result_Data_64_bytes_1[53];
	PlcInputs.ST70_1_DM260_PB_Result_Data_64_bytes_1[54] := HwInputs.ST70_1_DM260_PB_Result_Data_64_bytes_1[54];
	PlcInputs.ST70_1_DM260_PB_Result_Data_64_bytes_1[55] := HwInputs.ST70_1_DM260_PB_Result_Data_64_bytes_1[55];
	PlcInputs.ST70_1_DM260_PB_Result_Data_64_bytes_1[56] := HwInputs.ST70_1_DM260_PB_Result_Data_64_bytes_1[56];
	PlcInputs.ST70_1_DM260_PB_Result_Data_64_bytes_1[57] := HwInputs.ST70_1_DM260_PB_Result_Data_64_bytes_1[57];
	PlcInputs.ST70_1_DM260_PB_Result_Data_64_bytes_1[58] := HwInputs.ST70_1_DM260_PB_Result_Data_64_bytes_1[58];
	PlcInputs.ST70_1_DM260_PB_Result_Data_64_bytes_1[59] := HwInputs.ST70_1_DM260_PB_Result_Data_64_bytes_1[59];
	PlcInputs.ST70_1_DM260_PB_Result_Data_64_bytes_1[60] := HwInputs.ST70_1_DM260_PB_Result_Data_64_bytes_1[60];
	PlcInputs.ST70_1_DM260_PB_Result_Data_64_bytes_1[61] := HwInputs.ST70_1_DM260_PB_Result_Data_64_bytes_1[61];
	PlcInputs.ST70_1_DM260_PB_Result_Data_64_bytes_1[62] := HwInputs.ST70_1_DM260_PB_Result_Data_64_bytes_1[62];
	PlcInputs.ST70_1_DM260_PB_Result_Data_64_bytes_1[63] := HwInputs.ST70_1_DM260_PB_Result_Data_64_bytes_1[63];
	PlcInputs.ST70_1_DM260_PB_Result_Data_64_bytes_1[64] := HwInputs.ST70_1_DM260_PB_Result_Data_64_bytes_1[64];
	PlcInputs.ST70_1_DM260_PB_Result_Data_64_bytes_1[65] := HwInputs.ST70_1_DM260_PB_Result_Data_64_bytes_1[65];
	PlcInputs.ST70_1_DM260_PB_Result_Data_64_bytes_1[66] := HwInputs.ST70_1_DM260_PB_Result_Data_64_bytes_1[66];
	PlcInputs.ST70_1_DM260_PB_Result_Data_64_bytes_1[67] := HwInputs.ST70_1_DM260_PB_Result_Data_64_bytes_1[67];
	PlcInputs.ST70_1_DM260_PB_Result_Data_64_bytes_1[68] := HwInputs.ST70_1_DM260_PB_Result_Data_64_bytes_1[68];
	PlcInputs.ST70_1_DM260_PB_Result_Data_64_bytes_1[69] := HwInputs.ST70_1_DM260_PB_Result_Data_64_bytes_1[69];
	PlcInputs.ST70_1_DM260_PB_Result_Data_64_bytes_1[70] := HwInputs.ST70_1_DM260_PB_Result_Data_64_bytes_1[70];
	PlcInputs.ST70_1_DM260_PB_Result_Data_64_bytes_1[71] := HwInputs.ST70_1_DM260_PB_Result_Data_64_bytes_1[71];
	PlcInputs.ST70_2_DM260_PB_Acquisition_Status_1[0] := HwInputs.ST70_2_DM260_PB_Acquisition_Status_1[0];
	PlcInputs.ST70_2_DM260_PB_Acquisition_Status_1[1] := HwInputs.ST70_2_DM260_PB_Acquisition_Status_1[1];
	PlcInputs.ST70_2_DM260_PB_Acquisition_Status_1[2] := HwInputs.ST70_2_DM260_PB_Acquisition_Status_1[2];
	PlcInputs.ST70_2_DM260_PB_Results_Status_1 := HwInputs.ST70_2_DM260_PB_Results_Status_1;
	PlcInputs.ST70_2_DM260_PB_Soft_Event_Control_1 := HwInputs.ST70_2_DM260_PB_Soft_Event_Control_1;
	PlcInputs.ST70_2_DM260_PB_Result_Data_64_bytes_1[0] := HwInputs.ST70_2_DM260_PB_Result_Data_64_bytes_1[0];
	PlcInputs.ST70_2_DM260_PB_Result_Data_64_bytes_1[1] := HwInputs.ST70_2_DM260_PB_Result_Data_64_bytes_1[1];
	PlcInputs.ST70_2_DM260_PB_Result_Data_64_bytes_1[2] := HwInputs.ST70_2_DM260_PB_Result_Data_64_bytes_1[2];
	PlcInputs.ST70_2_DM260_PB_Result_Data_64_bytes_1[3] := HwInputs.ST70_2_DM260_PB_Result_Data_64_bytes_1[3];
	PlcInputs.ST70_2_DM260_PB_Result_Data_64_bytes_1[4] := HwInputs.ST70_2_DM260_PB_Result_Data_64_bytes_1[4];
	PlcInputs.ST70_2_DM260_PB_Result_Data_64_bytes_1[5] := HwInputs.ST70_2_DM260_PB_Result_Data_64_bytes_1[5];
	PlcInputs.ST70_2_DM260_PB_Result_Data_64_bytes_1[6] := HwInputs.ST70_2_DM260_PB_Result_Data_64_bytes_1[6];
	PlcInputs.ST70_2_DM260_PB_Result_Data_64_bytes_1[7] := HwInputs.ST70_2_DM260_PB_Result_Data_64_bytes_1[7];
	PlcInputs.ST70_2_DM260_PB_Result_Data_64_bytes_1[8] := HwInputs.ST70_2_DM260_PB_Result_Data_64_bytes_1[8];
	PlcInputs.ST70_2_DM260_PB_Result_Data_64_bytes_1[9] := HwInputs.ST70_2_DM260_PB_Result_Data_64_bytes_1[9];
	PlcInputs.ST70_2_DM260_PB_Result_Data_64_bytes_1[10] := HwInputs.ST70_2_DM260_PB_Result_Data_64_bytes_1[10];
	PlcInputs.ST70_2_DM260_PB_Result_Data_64_bytes_1[11] := HwInputs.ST70_2_DM260_PB_Result_Data_64_bytes_1[11];
	PlcInputs.ST70_2_DM260_PB_Result_Data_64_bytes_1[12] := HwInputs.ST70_2_DM260_PB_Result_Data_64_bytes_1[12];
	PlcInputs.ST70_2_DM260_PB_Result_Data_64_bytes_1[13] := HwInputs.ST70_2_DM260_PB_Result_Data_64_bytes_1[13];
	PlcInputs.ST70_2_DM260_PB_Result_Data_64_bytes_1[14] := HwInputs.ST70_2_DM260_PB_Result_Data_64_bytes_1[14];
	PlcInputs.ST70_2_DM260_PB_Result_Data_64_bytes_1[15] := HwInputs.ST70_2_DM260_PB_Result_Data_64_bytes_1[15];
	PlcInputs.ST70_2_DM260_PB_Result_Data_64_bytes_1[16] := HwInputs.ST70_2_DM260_PB_Result_Data_64_bytes_1[16];
	PlcInputs.ST70_2_DM260_PB_Result_Data_64_bytes_1[17] := HwInputs.ST70_2_DM260_PB_Result_Data_64_bytes_1[17];
	PlcInputs.ST70_2_DM260_PB_Result_Data_64_bytes_1[18] := HwInputs.ST70_2_DM260_PB_Result_Data_64_bytes_1[18];
	PlcInputs.ST70_2_DM260_PB_Result_Data_64_bytes_1[19] := HwInputs.ST70_2_DM260_PB_Result_Data_64_bytes_1[19];
	PlcInputs.ST70_2_DM260_PB_Result_Data_64_bytes_1[20] := HwInputs.ST70_2_DM260_PB_Result_Data_64_bytes_1[20];
	PlcInputs.ST70_2_DM260_PB_Result_Data_64_bytes_1[21] := HwInputs.ST70_2_DM260_PB_Result_Data_64_bytes_1[21];
	PlcInputs.ST70_2_DM260_PB_Result_Data_64_bytes_1[22] := HwInputs.ST70_2_DM260_PB_Result_Data_64_bytes_1[22];
	PlcInputs.ST70_2_DM260_PB_Result_Data_64_bytes_1[23] := HwInputs.ST70_2_DM260_PB_Result_Data_64_bytes_1[23];
	PlcInputs.ST70_2_DM260_PB_Result_Data_64_bytes_1[24] := HwInputs.ST70_2_DM260_PB_Result_Data_64_bytes_1[24];
	PlcInputs.ST70_2_DM260_PB_Result_Data_64_bytes_1[25] := HwInputs.ST70_2_DM260_PB_Result_Data_64_bytes_1[25];
	PlcInputs.ST70_2_DM260_PB_Result_Data_64_bytes_1[26] := HwInputs.ST70_2_DM260_PB_Result_Data_64_bytes_1[26];
	PlcInputs.ST70_2_DM260_PB_Result_Data_64_bytes_1[27] := HwInputs.ST70_2_DM260_PB_Result_Data_64_bytes_1[27];
	PlcInputs.ST70_2_DM260_PB_Result_Data_64_bytes_1[28] := HwInputs.ST70_2_DM260_PB_Result_Data_64_bytes_1[28];
	PlcInputs.ST70_2_DM260_PB_Result_Data_64_bytes_1[29] := HwInputs.ST70_2_DM260_PB_Result_Data_64_bytes_1[29];
	PlcInputs.ST70_2_DM260_PB_Result_Data_64_bytes_1[30] := HwInputs.ST70_2_DM260_PB_Result_Data_64_bytes_1[30];
	PlcInputs.ST70_2_DM260_PB_Result_Data_64_bytes_1[31] := HwInputs.ST70_2_DM260_PB_Result_Data_64_bytes_1[31];
	PlcInputs.ST70_2_DM260_PB_Result_Data_64_bytes_1[32] := HwInputs.ST70_2_DM260_PB_Result_Data_64_bytes_1[32];
	PlcInputs.ST70_2_DM260_PB_Result_Data_64_bytes_1[33] := HwInputs.ST70_2_DM260_PB_Result_Data_64_bytes_1[33];
	PlcInputs.ST70_2_DM260_PB_Result_Data_64_bytes_1[34] := HwInputs.ST70_2_DM260_PB_Result_Data_64_bytes_1[34];
	PlcInputs.ST70_2_DM260_PB_Result_Data_64_bytes_1[35] := HwInputs.ST70_2_DM260_PB_Result_Data_64_bytes_1[35];
	PlcInputs.ST70_2_DM260_PB_Result_Data_64_bytes_1[36] := HwInputs.ST70_2_DM260_PB_Result_Data_64_bytes_1[36];
	PlcInputs.ST70_2_DM260_PB_Result_Data_64_bytes_1[37] := HwInputs.ST70_2_DM260_PB_Result_Data_64_bytes_1[37];
	PlcInputs.ST70_2_DM260_PB_Result_Data_64_bytes_1[38] := HwInputs.ST70_2_DM260_PB_Result_Data_64_bytes_1[38];
	PlcInputs.ST70_2_DM260_PB_Result_Data_64_bytes_1[39] := HwInputs.ST70_2_DM260_PB_Result_Data_64_bytes_1[39];
	PlcInputs.ST70_2_DM260_PB_Result_Data_64_bytes_1[40] := HwInputs.ST70_2_DM260_PB_Result_Data_64_bytes_1[40];
	PlcInputs.ST70_2_DM260_PB_Result_Data_64_bytes_1[41] := HwInputs.ST70_2_DM260_PB_Result_Data_64_bytes_1[41];
	PlcInputs.ST70_2_DM260_PB_Result_Data_64_bytes_1[42] := HwInputs.ST70_2_DM260_PB_Result_Data_64_bytes_1[42];
	PlcInputs.ST70_2_DM260_PB_Result_Data_64_bytes_1[43] := HwInputs.ST70_2_DM260_PB_Result_Data_64_bytes_1[43];
	PlcInputs.ST70_2_DM260_PB_Result_Data_64_bytes_1[44] := HwInputs.ST70_2_DM260_PB_Result_Data_64_bytes_1[44];
	PlcInputs.ST70_2_DM260_PB_Result_Data_64_bytes_1[45] := HwInputs.ST70_2_DM260_PB_Result_Data_64_bytes_1[45];
	PlcInputs.ST70_2_DM260_PB_Result_Data_64_bytes_1[46] := HwInputs.ST70_2_DM260_PB_Result_Data_64_bytes_1[46];
	PlcInputs.ST70_2_DM260_PB_Result_Data_64_bytes_1[47] := HwInputs.ST70_2_DM260_PB_Result_Data_64_bytes_1[47];
	PlcInputs.ST70_2_DM260_PB_Result_Data_64_bytes_1[48] := HwInputs.ST70_2_DM260_PB_Result_Data_64_bytes_1[48];
	PlcInputs.ST70_2_DM260_PB_Result_Data_64_bytes_1[49] := HwInputs.ST70_2_DM260_PB_Result_Data_64_bytes_1[49];
	PlcInputs.ST70_2_DM260_PB_Result_Data_64_bytes_1[50] := HwInputs.ST70_2_DM260_PB_Result_Data_64_bytes_1[50];
	PlcInputs.ST70_2_DM260_PB_Result_Data_64_bytes_1[51] := HwInputs.ST70_2_DM260_PB_Result_Data_64_bytes_1[51];
	PlcInputs.ST70_2_DM260_PB_Result_Data_64_bytes_1[52] := HwInputs.ST70_2_DM260_PB_Result_Data_64_bytes_1[52];
	PlcInputs.ST70_2_DM260_PB_Result_Data_64_bytes_1[53] := HwInputs.ST70_2_DM260_PB_Result_Data_64_bytes_1[53];
	PlcInputs.ST70_2_DM260_PB_Result_Data_64_bytes_1[54] := HwInputs.ST70_2_DM260_PB_Result_Data_64_bytes_1[54];
	PlcInputs.ST70_2_DM260_PB_Result_Data_64_bytes_1[55] := HwInputs.ST70_2_DM260_PB_Result_Data_64_bytes_1[55];
	PlcInputs.ST70_2_DM260_PB_Result_Data_64_bytes_1[56] := HwInputs.ST70_2_DM260_PB_Result_Data_64_bytes_1[56];
	PlcInputs.ST70_2_DM260_PB_Result_Data_64_bytes_1[57] := HwInputs.ST70_2_DM260_PB_Result_Data_64_bytes_1[57];
	PlcInputs.ST70_2_DM260_PB_Result_Data_64_bytes_1[58] := HwInputs.ST70_2_DM260_PB_Result_Data_64_bytes_1[58];
	PlcInputs.ST70_2_DM260_PB_Result_Data_64_bytes_1[59] := HwInputs.ST70_2_DM260_PB_Result_Data_64_bytes_1[59];
	PlcInputs.ST70_2_DM260_PB_Result_Data_64_bytes_1[60] := HwInputs.ST70_2_DM260_PB_Result_Data_64_bytes_1[60];
	PlcInputs.ST70_2_DM260_PB_Result_Data_64_bytes_1[61] := HwInputs.ST70_2_DM260_PB_Result_Data_64_bytes_1[61];
	PlcInputs.ST70_2_DM260_PB_Result_Data_64_bytes_1[62] := HwInputs.ST70_2_DM260_PB_Result_Data_64_bytes_1[62];
	PlcInputs.ST70_2_DM260_PB_Result_Data_64_bytes_1[63] := HwInputs.ST70_2_DM260_PB_Result_Data_64_bytes_1[63];
	PlcInputs.ST70_2_DM260_PB_Result_Data_64_bytes_1[64] := HwInputs.ST70_2_DM260_PB_Result_Data_64_bytes_1[64];
	PlcInputs.ST70_2_DM260_PB_Result_Data_64_bytes_1[65] := HwInputs.ST70_2_DM260_PB_Result_Data_64_bytes_1[65];
	PlcInputs.ST70_2_DM260_PB_Result_Data_64_bytes_1[66] := HwInputs.ST70_2_DM260_PB_Result_Data_64_bytes_1[66];
	PlcInputs.ST70_2_DM260_PB_Result_Data_64_bytes_1[67] := HwInputs.ST70_2_DM260_PB_Result_Data_64_bytes_1[67];
	PlcInputs.ST70_2_DM260_PB_Result_Data_64_bytes_1[68] := HwInputs.ST70_2_DM260_PB_Result_Data_64_bytes_1[68];
	PlcInputs.ST70_2_DM260_PB_Result_Data_64_bytes_1[69] := HwInputs.ST70_2_DM260_PB_Result_Data_64_bytes_1[69];
	PlcInputs.ST70_2_DM260_PB_Result_Data_64_bytes_1[70] := HwInputs.ST70_2_DM260_PB_Result_Data_64_bytes_1[70];
	PlcInputs.ST70_2_DM260_PB_Result_Data_64_bytes_1[71] := HwInputs.ST70_2_DM260_PB_Result_Data_64_bytes_1[71];
	PlcInputs.ST70_1_CMMT_3GF1_DO_SERVO_1_Siemens_telegram_111_PZD_12_12[0] := HwInputs.ST70_1_CMMT_3GF1_DO_SERVO_1_Siemens_telegram_111_PZD_12_12[0];
	PlcInputs.ST70_1_CMMT_3GF1_DO_SERVO_1_Siemens_telegram_111_PZD_12_12[1] := HwInputs.ST70_1_CMMT_3GF1_DO_SERVO_1_Siemens_telegram_111_PZD_12_12[1];
	PlcInputs.ST70_1_CMMT_3GF1_DO_SERVO_1_Siemens_telegram_111_PZD_12_12[2] := HwInputs.ST70_1_CMMT_3GF1_DO_SERVO_1_Siemens_telegram_111_PZD_12_12[2];
	PlcInputs.ST70_1_CMMT_3GF1_DO_SERVO_1_Siemens_telegram_111_PZD_12_12[3] := HwInputs.ST70_1_CMMT_3GF1_DO_SERVO_1_Siemens_telegram_111_PZD_12_12[3];
	PlcInputs.ST70_1_CMMT_3GF1_DO_SERVO_1_Siemens_telegram_111_PZD_12_12[4] := HwInputs.ST70_1_CMMT_3GF1_DO_SERVO_1_Siemens_telegram_111_PZD_12_12[4];
	PlcInputs.ST70_1_CMMT_3GF1_DO_SERVO_1_Siemens_telegram_111_PZD_12_12[5] := HwInputs.ST70_1_CMMT_3GF1_DO_SERVO_1_Siemens_telegram_111_PZD_12_12[5];
	PlcInputs.ST70_1_CMMT_3GF1_DO_SERVO_1_Siemens_telegram_111_PZD_12_12[6] := HwInputs.ST70_1_CMMT_3GF1_DO_SERVO_1_Siemens_telegram_111_PZD_12_12[6];
	PlcInputs.ST70_1_CMMT_3GF1_DO_SERVO_1_Siemens_telegram_111_PZD_12_12[7] := HwInputs.ST70_1_CMMT_3GF1_DO_SERVO_1_Siemens_telegram_111_PZD_12_12[7];
	PlcInputs.ST70_1_CMMT_3GF1_DO_SERVO_1_Siemens_telegram_111_PZD_12_12[8] := HwInputs.ST70_1_CMMT_3GF1_DO_SERVO_1_Siemens_telegram_111_PZD_12_12[8];
	PlcInputs.ST70_1_CMMT_3GF1_DO_SERVO_1_Siemens_telegram_111_PZD_12_12[9] := HwInputs.ST70_1_CMMT_3GF1_DO_SERVO_1_Siemens_telegram_111_PZD_12_12[9];
	PlcInputs.ST70_1_CMMT_3GF1_DO_SERVO_1_Siemens_telegram_111_PZD_12_12[10] := HwInputs.ST70_1_CMMT_3GF1_DO_SERVO_1_Siemens_telegram_111_PZD_12_12[10];
	PlcInputs.ST70_1_CMMT_3GF1_DO_SERVO_1_Siemens_telegram_111_PZD_12_12[11] := HwInputs.ST70_1_CMMT_3GF1_DO_SERVO_1_Siemens_telegram_111_PZD_12_12[11];
	PlcInputs.ST70_1_CMMT_3GF1_DO_SERVO_1_Siemens_telegram_111_PZD_12_12[12] := HwInputs.ST70_1_CMMT_3GF1_DO_SERVO_1_Siemens_telegram_111_PZD_12_12[12];
	PlcInputs.ST70_1_CMMT_3GF1_DO_SERVO_1_Siemens_telegram_111_PZD_12_12[13] := HwInputs.ST70_1_CMMT_3GF1_DO_SERVO_1_Siemens_telegram_111_PZD_12_12[13];
	PlcInputs.ST70_1_CMMT_3GF1_DO_SERVO_1_Siemens_telegram_111_PZD_12_12[14] := HwInputs.ST70_1_CMMT_3GF1_DO_SERVO_1_Siemens_telegram_111_PZD_12_12[14];
	PlcInputs.ST70_1_CMMT_3GF1_DO_SERVO_1_Siemens_telegram_111_PZD_12_12[15] := HwInputs.ST70_1_CMMT_3GF1_DO_SERVO_1_Siemens_telegram_111_PZD_12_12[15];
	PlcInputs.ST70_1_CMMT_3GF1_DO_SERVO_1_Siemens_telegram_111_PZD_12_12[16] := HwInputs.ST70_1_CMMT_3GF1_DO_SERVO_1_Siemens_telegram_111_PZD_12_12[16];
	PlcInputs.ST70_1_CMMT_3GF1_DO_SERVO_1_Siemens_telegram_111_PZD_12_12[17] := HwInputs.ST70_1_CMMT_3GF1_DO_SERVO_1_Siemens_telegram_111_PZD_12_12[17];
	PlcInputs.ST70_1_CMMT_3GF1_DO_SERVO_1_Siemens_telegram_111_PZD_12_12[18] := HwInputs.ST70_1_CMMT_3GF1_DO_SERVO_1_Siemens_telegram_111_PZD_12_12[18];
	PlcInputs.ST70_1_CMMT_3GF1_DO_SERVO_1_Siemens_telegram_111_PZD_12_12[19] := HwInputs.ST70_1_CMMT_3GF1_DO_SERVO_1_Siemens_telegram_111_PZD_12_12[19];
	PlcInputs.ST70_1_CMMT_3GF1_DO_SERVO_1_Siemens_telegram_111_PZD_12_12[20] := HwInputs.ST70_1_CMMT_3GF1_DO_SERVO_1_Siemens_telegram_111_PZD_12_12[20];
	PlcInputs.ST70_1_CMMT_3GF1_DO_SERVO_1_Siemens_telegram_111_PZD_12_12[21] := HwInputs.ST70_1_CMMT_3GF1_DO_SERVO_1_Siemens_telegram_111_PZD_12_12[21];
	PlcInputs.ST70_1_CMMT_3GF1_DO_SERVO_1_Siemens_telegram_111_PZD_12_12[22] := HwInputs.ST70_1_CMMT_3GF1_DO_SERVO_1_Siemens_telegram_111_PZD_12_12[22];
	PlcInputs.ST70_1_CMMT_3GF1_DO_SERVO_1_Siemens_telegram_111_PZD_12_12[23] := HwInputs.ST70_1_CMMT_3GF1_DO_SERVO_1_Siemens_telegram_111_PZD_12_12[23];
	PlcInputs.ST70_1_CMMT_3GF2_DO_SERVO_1_Siemens_telegram_111_PZD_12_12[0] := HwInputs.ST70_1_CMMT_3GF2_DO_SERVO_1_Siemens_telegram_111_PZD_12_12[0];
	PlcInputs.ST70_1_CMMT_3GF2_DO_SERVO_1_Siemens_telegram_111_PZD_12_12[1] := HwInputs.ST70_1_CMMT_3GF2_DO_SERVO_1_Siemens_telegram_111_PZD_12_12[1];
	PlcInputs.ST70_1_CMMT_3GF2_DO_SERVO_1_Siemens_telegram_111_PZD_12_12[2] := HwInputs.ST70_1_CMMT_3GF2_DO_SERVO_1_Siemens_telegram_111_PZD_12_12[2];
	PlcInputs.ST70_1_CMMT_3GF2_DO_SERVO_1_Siemens_telegram_111_PZD_12_12[3] := HwInputs.ST70_1_CMMT_3GF2_DO_SERVO_1_Siemens_telegram_111_PZD_12_12[3];
	PlcInputs.ST70_1_CMMT_3GF2_DO_SERVO_1_Siemens_telegram_111_PZD_12_12[4] := HwInputs.ST70_1_CMMT_3GF2_DO_SERVO_1_Siemens_telegram_111_PZD_12_12[4];
	PlcInputs.ST70_1_CMMT_3GF2_DO_SERVO_1_Siemens_telegram_111_PZD_12_12[5] := HwInputs.ST70_1_CMMT_3GF2_DO_SERVO_1_Siemens_telegram_111_PZD_12_12[5];
	PlcInputs.ST70_1_CMMT_3GF2_DO_SERVO_1_Siemens_telegram_111_PZD_12_12[6] := HwInputs.ST70_1_CMMT_3GF2_DO_SERVO_1_Siemens_telegram_111_PZD_12_12[6];
	PlcInputs.ST70_1_CMMT_3GF2_DO_SERVO_1_Siemens_telegram_111_PZD_12_12[7] := HwInputs.ST70_1_CMMT_3GF2_DO_SERVO_1_Siemens_telegram_111_PZD_12_12[7];
	PlcInputs.ST70_1_CMMT_3GF2_DO_SERVO_1_Siemens_telegram_111_PZD_12_12[8] := HwInputs.ST70_1_CMMT_3GF2_DO_SERVO_1_Siemens_telegram_111_PZD_12_12[8];
	PlcInputs.ST70_1_CMMT_3GF2_DO_SERVO_1_Siemens_telegram_111_PZD_12_12[9] := HwInputs.ST70_1_CMMT_3GF2_DO_SERVO_1_Siemens_telegram_111_PZD_12_12[9];
	PlcInputs.ST70_1_CMMT_3GF2_DO_SERVO_1_Siemens_telegram_111_PZD_12_12[10] := HwInputs.ST70_1_CMMT_3GF2_DO_SERVO_1_Siemens_telegram_111_PZD_12_12[10];
	PlcInputs.ST70_1_CMMT_3GF2_DO_SERVO_1_Siemens_telegram_111_PZD_12_12[11] := HwInputs.ST70_1_CMMT_3GF2_DO_SERVO_1_Siemens_telegram_111_PZD_12_12[11];
	PlcInputs.ST70_1_CMMT_3GF2_DO_SERVO_1_Siemens_telegram_111_PZD_12_12[12] := HwInputs.ST70_1_CMMT_3GF2_DO_SERVO_1_Siemens_telegram_111_PZD_12_12[12];
	PlcInputs.ST70_1_CMMT_3GF2_DO_SERVO_1_Siemens_telegram_111_PZD_12_12[13] := HwInputs.ST70_1_CMMT_3GF2_DO_SERVO_1_Siemens_telegram_111_PZD_12_12[13];
	PlcInputs.ST70_1_CMMT_3GF2_DO_SERVO_1_Siemens_telegram_111_PZD_12_12[14] := HwInputs.ST70_1_CMMT_3GF2_DO_SERVO_1_Siemens_telegram_111_PZD_12_12[14];
	PlcInputs.ST70_1_CMMT_3GF2_DO_SERVO_1_Siemens_telegram_111_PZD_12_12[15] := HwInputs.ST70_1_CMMT_3GF2_DO_SERVO_1_Siemens_telegram_111_PZD_12_12[15];
	PlcInputs.ST70_1_CMMT_3GF2_DO_SERVO_1_Siemens_telegram_111_PZD_12_12[16] := HwInputs.ST70_1_CMMT_3GF2_DO_SERVO_1_Siemens_telegram_111_PZD_12_12[16];
	PlcInputs.ST70_1_CMMT_3GF2_DO_SERVO_1_Siemens_telegram_111_PZD_12_12[17] := HwInputs.ST70_1_CMMT_3GF2_DO_SERVO_1_Siemens_telegram_111_PZD_12_12[17];
	PlcInputs.ST70_1_CMMT_3GF2_DO_SERVO_1_Siemens_telegram_111_PZD_12_12[18] := HwInputs.ST70_1_CMMT_3GF2_DO_SERVO_1_Siemens_telegram_111_PZD_12_12[18];
	PlcInputs.ST70_1_CMMT_3GF2_DO_SERVO_1_Siemens_telegram_111_PZD_12_12[19] := HwInputs.ST70_1_CMMT_3GF2_DO_SERVO_1_Siemens_telegram_111_PZD_12_12[19];
	PlcInputs.ST70_1_CMMT_3GF2_DO_SERVO_1_Siemens_telegram_111_PZD_12_12[20] := HwInputs.ST70_1_CMMT_3GF2_DO_SERVO_1_Siemens_telegram_111_PZD_12_12[20];
	PlcInputs.ST70_1_CMMT_3GF2_DO_SERVO_1_Siemens_telegram_111_PZD_12_12[21] := HwInputs.ST70_1_CMMT_3GF2_DO_SERVO_1_Siemens_telegram_111_PZD_12_12[21];
	PlcInputs.ST70_1_CMMT_3GF2_DO_SERVO_1_Siemens_telegram_111_PZD_12_12[22] := HwInputs.ST70_1_CMMT_3GF2_DO_SERVO_1_Siemens_telegram_111_PZD_12_12[22];
	PlcInputs.ST70_1_CMMT_3GF2_DO_SERVO_1_Siemens_telegram_111_PZD_12_12[23] := HwInputs.ST70_1_CMMT_3GF2_DO_SERVO_1_Siemens_telegram_111_PZD_12_12[23];
	PlcInputs.ST70_3_DM260_PB_Acquisition_Status_1[0] := HwInputs.ST70_3_DM260_PB_Acquisition_Status_1[0];
	PlcInputs.ST70_3_DM260_PB_Acquisition_Status_1[1] := HwInputs.ST70_3_DM260_PB_Acquisition_Status_1[1];
	PlcInputs.ST70_3_DM260_PB_Acquisition_Status_1[2] := HwInputs.ST70_3_DM260_PB_Acquisition_Status_1[2];
	PlcInputs.ST70_3_DM260_PB_Results_Status_1 := HwInputs.ST70_3_DM260_PB_Results_Status_1;
	PlcInputs.ST70_3_DM260_PB_Soft_Event_Control_1 := HwInputs.ST70_3_DM260_PB_Soft_Event_Control_1;
	PlcInputs.ST70_3_DM260_PB_Result_Data_64_bytes_1[0] := HwInputs.ST70_3_DM260_PB_Result_Data_64_bytes_1[0];
	PlcInputs.ST70_3_DM260_PB_Result_Data_64_bytes_1[1] := HwInputs.ST70_3_DM260_PB_Result_Data_64_bytes_1[1];
	PlcInputs.ST70_3_DM260_PB_Result_Data_64_bytes_1[2] := HwInputs.ST70_3_DM260_PB_Result_Data_64_bytes_1[2];
	PlcInputs.ST70_3_DM260_PB_Result_Data_64_bytes_1[3] := HwInputs.ST70_3_DM260_PB_Result_Data_64_bytes_1[3];
	PlcInputs.ST70_3_DM260_PB_Result_Data_64_bytes_1[4] := HwInputs.ST70_3_DM260_PB_Result_Data_64_bytes_1[4];
	PlcInputs.ST70_3_DM260_PB_Result_Data_64_bytes_1[5] := HwInputs.ST70_3_DM260_PB_Result_Data_64_bytes_1[5];
	PlcInputs.ST70_3_DM260_PB_Result_Data_64_bytes_1[6] := HwInputs.ST70_3_DM260_PB_Result_Data_64_bytes_1[6];
	PlcInputs.ST70_3_DM260_PB_Result_Data_64_bytes_1[7] := HwInputs.ST70_3_DM260_PB_Result_Data_64_bytes_1[7];
	PlcInputs.ST70_3_DM260_PB_Result_Data_64_bytes_1[8] := HwInputs.ST70_3_DM260_PB_Result_Data_64_bytes_1[8];
	PlcInputs.ST70_3_DM260_PB_Result_Data_64_bytes_1[9] := HwInputs.ST70_3_DM260_PB_Result_Data_64_bytes_1[9];
	PlcInputs.ST70_3_DM260_PB_Result_Data_64_bytes_1[10] := HwInputs.ST70_3_DM260_PB_Result_Data_64_bytes_1[10];
	PlcInputs.ST70_3_DM260_PB_Result_Data_64_bytes_1[11] := HwInputs.ST70_3_DM260_PB_Result_Data_64_bytes_1[11];
	PlcInputs.ST70_3_DM260_PB_Result_Data_64_bytes_1[12] := HwInputs.ST70_3_DM260_PB_Result_Data_64_bytes_1[12];
	PlcInputs.ST70_3_DM260_PB_Result_Data_64_bytes_1[13] := HwInputs.ST70_3_DM260_PB_Result_Data_64_bytes_1[13];
	PlcInputs.ST70_3_DM260_PB_Result_Data_64_bytes_1[14] := HwInputs.ST70_3_DM260_PB_Result_Data_64_bytes_1[14];
	PlcInputs.ST70_3_DM260_PB_Result_Data_64_bytes_1[15] := HwInputs.ST70_3_DM260_PB_Result_Data_64_bytes_1[15];
	PlcInputs.ST70_3_DM260_PB_Result_Data_64_bytes_1[16] := HwInputs.ST70_3_DM260_PB_Result_Data_64_bytes_1[16];
	PlcInputs.ST70_3_DM260_PB_Result_Data_64_bytes_1[17] := HwInputs.ST70_3_DM260_PB_Result_Data_64_bytes_1[17];
	PlcInputs.ST70_3_DM260_PB_Result_Data_64_bytes_1[18] := HwInputs.ST70_3_DM260_PB_Result_Data_64_bytes_1[18];
	PlcInputs.ST70_3_DM260_PB_Result_Data_64_bytes_1[19] := HwInputs.ST70_3_DM260_PB_Result_Data_64_bytes_1[19];
	PlcInputs.ST70_3_DM260_PB_Result_Data_64_bytes_1[20] := HwInputs.ST70_3_DM260_PB_Result_Data_64_bytes_1[20];
	PlcInputs.ST70_3_DM260_PB_Result_Data_64_bytes_1[21] := HwInputs.ST70_3_DM260_PB_Result_Data_64_bytes_1[21];
	PlcInputs.ST70_3_DM260_PB_Result_Data_64_bytes_1[22] := HwInputs.ST70_3_DM260_PB_Result_Data_64_bytes_1[22];
	PlcInputs.ST70_3_DM260_PB_Result_Data_64_bytes_1[23] := HwInputs.ST70_3_DM260_PB_Result_Data_64_bytes_1[23];
	PlcInputs.ST70_3_DM260_PB_Result_Data_64_bytes_1[24] := HwInputs.ST70_3_DM260_PB_Result_Data_64_bytes_1[24];
	PlcInputs.ST70_3_DM260_PB_Result_Data_64_bytes_1[25] := HwInputs.ST70_3_DM260_PB_Result_Data_64_bytes_1[25];
	PlcInputs.ST70_3_DM260_PB_Result_Data_64_bytes_1[26] := HwInputs.ST70_3_DM260_PB_Result_Data_64_bytes_1[26];
	PlcInputs.ST70_3_DM260_PB_Result_Data_64_bytes_1[27] := HwInputs.ST70_3_DM260_PB_Result_Data_64_bytes_1[27];
	PlcInputs.ST70_3_DM260_PB_Result_Data_64_bytes_1[28] := HwInputs.ST70_3_DM260_PB_Result_Data_64_bytes_1[28];
	PlcInputs.ST70_3_DM260_PB_Result_Data_64_bytes_1[29] := HwInputs.ST70_3_DM260_PB_Result_Data_64_bytes_1[29];
	PlcInputs.ST70_3_DM260_PB_Result_Data_64_bytes_1[30] := HwInputs.ST70_3_DM260_PB_Result_Data_64_bytes_1[30];
	PlcInputs.ST70_3_DM260_PB_Result_Data_64_bytes_1[31] := HwInputs.ST70_3_DM260_PB_Result_Data_64_bytes_1[31];
	PlcInputs.ST70_3_DM260_PB_Result_Data_64_bytes_1[32] := HwInputs.ST70_3_DM260_PB_Result_Data_64_bytes_1[32];
	PlcInputs.ST70_3_DM260_PB_Result_Data_64_bytes_1[33] := HwInputs.ST70_3_DM260_PB_Result_Data_64_bytes_1[33];
	PlcInputs.ST70_3_DM260_PB_Result_Data_64_bytes_1[34] := HwInputs.ST70_3_DM260_PB_Result_Data_64_bytes_1[34];
	PlcInputs.ST70_3_DM260_PB_Result_Data_64_bytes_1[35] := HwInputs.ST70_3_DM260_PB_Result_Data_64_bytes_1[35];
	PlcInputs.ST70_3_DM260_PB_Result_Data_64_bytes_1[36] := HwInputs.ST70_3_DM260_PB_Result_Data_64_bytes_1[36];
	PlcInputs.ST70_3_DM260_PB_Result_Data_64_bytes_1[37] := HwInputs.ST70_3_DM260_PB_Result_Data_64_bytes_1[37];
	PlcInputs.ST70_3_DM260_PB_Result_Data_64_bytes_1[38] := HwInputs.ST70_3_DM260_PB_Result_Data_64_bytes_1[38];
	PlcInputs.ST70_3_DM260_PB_Result_Data_64_bytes_1[39] := HwInputs.ST70_3_DM260_PB_Result_Data_64_bytes_1[39];
	PlcInputs.ST70_3_DM260_PB_Result_Data_64_bytes_1[40] := HwInputs.ST70_3_DM260_PB_Result_Data_64_bytes_1[40];
	PlcInputs.ST70_3_DM260_PB_Result_Data_64_bytes_1[41] := HwInputs.ST70_3_DM260_PB_Result_Data_64_bytes_1[41];
	PlcInputs.ST70_3_DM260_PB_Result_Data_64_bytes_1[42] := HwInputs.ST70_3_DM260_PB_Result_Data_64_bytes_1[42];
	PlcInputs.ST70_3_DM260_PB_Result_Data_64_bytes_1[43] := HwInputs.ST70_3_DM260_PB_Result_Data_64_bytes_1[43];
	PlcInputs.ST70_3_DM260_PB_Result_Data_64_bytes_1[44] := HwInputs.ST70_3_DM260_PB_Result_Data_64_bytes_1[44];
	PlcInputs.ST70_3_DM260_PB_Result_Data_64_bytes_1[45] := HwInputs.ST70_3_DM260_PB_Result_Data_64_bytes_1[45];
	PlcInputs.ST70_3_DM260_PB_Result_Data_64_bytes_1[46] := HwInputs.ST70_3_DM260_PB_Result_Data_64_bytes_1[46];
	PlcInputs.ST70_3_DM260_PB_Result_Data_64_bytes_1[47] := HwInputs.ST70_3_DM260_PB_Result_Data_64_bytes_1[47];
	PlcInputs.ST70_3_DM260_PB_Result_Data_64_bytes_1[48] := HwInputs.ST70_3_DM260_PB_Result_Data_64_bytes_1[48];
	PlcInputs.ST70_3_DM260_PB_Result_Data_64_bytes_1[49] := HwInputs.ST70_3_DM260_PB_Result_Data_64_bytes_1[49];
	PlcInputs.ST70_3_DM260_PB_Result_Data_64_bytes_1[50] := HwInputs.ST70_3_DM260_PB_Result_Data_64_bytes_1[50];
	PlcInputs.ST70_3_DM260_PB_Result_Data_64_bytes_1[51] := HwInputs.ST70_3_DM260_PB_Result_Data_64_bytes_1[51];
	PlcInputs.ST70_3_DM260_PB_Result_Data_64_bytes_1[52] := HwInputs.ST70_3_DM260_PB_Result_Data_64_bytes_1[52];
	PlcInputs.ST70_3_DM260_PB_Result_Data_64_bytes_1[53] := HwInputs.ST70_3_DM260_PB_Result_Data_64_bytes_1[53];
	PlcInputs.ST70_3_DM260_PB_Result_Data_64_bytes_1[54] := HwInputs.ST70_3_DM260_PB_Result_Data_64_bytes_1[54];
	PlcInputs.ST70_3_DM260_PB_Result_Data_64_bytes_1[55] := HwInputs.ST70_3_DM260_PB_Result_Data_64_bytes_1[55];
	PlcInputs.ST70_3_DM260_PB_Result_Data_64_bytes_1[56] := HwInputs.ST70_3_DM260_PB_Result_Data_64_bytes_1[56];
	PlcInputs.ST70_3_DM260_PB_Result_Data_64_bytes_1[57] := HwInputs.ST70_3_DM260_PB_Result_Data_64_bytes_1[57];
	PlcInputs.ST70_3_DM260_PB_Result_Data_64_bytes_1[58] := HwInputs.ST70_3_DM260_PB_Result_Data_64_bytes_1[58];
	PlcInputs.ST70_3_DM260_PB_Result_Data_64_bytes_1[59] := HwInputs.ST70_3_DM260_PB_Result_Data_64_bytes_1[59];
	PlcInputs.ST70_3_DM260_PB_Result_Data_64_bytes_1[60] := HwInputs.ST70_3_DM260_PB_Result_Data_64_bytes_1[60];
	PlcInputs.ST70_3_DM260_PB_Result_Data_64_bytes_1[61] := HwInputs.ST70_3_DM260_PB_Result_Data_64_bytes_1[61];
	PlcInputs.ST70_3_DM260_PB_Result_Data_64_bytes_1[62] := HwInputs.ST70_3_DM260_PB_Result_Data_64_bytes_1[62];
	PlcInputs.ST70_3_DM260_PB_Result_Data_64_bytes_1[63] := HwInputs.ST70_3_DM260_PB_Result_Data_64_bytes_1[63];
	PlcInputs.ST70_3_DM260_PB_Result_Data_64_bytes_1[64] := HwInputs.ST70_3_DM260_PB_Result_Data_64_bytes_1[64];
	PlcInputs.ST70_3_DM260_PB_Result_Data_64_bytes_1[65] := HwInputs.ST70_3_DM260_PB_Result_Data_64_bytes_1[65];
	PlcInputs.ST70_3_DM260_PB_Result_Data_64_bytes_1[66] := HwInputs.ST70_3_DM260_PB_Result_Data_64_bytes_1[66];
	PlcInputs.ST70_3_DM260_PB_Result_Data_64_bytes_1[67] := HwInputs.ST70_3_DM260_PB_Result_Data_64_bytes_1[67];
	PlcInputs.ST70_3_DM260_PB_Result_Data_64_bytes_1[68] := HwInputs.ST70_3_DM260_PB_Result_Data_64_bytes_1[68];
	PlcInputs.ST70_3_DM260_PB_Result_Data_64_bytes_1[69] := HwInputs.ST70_3_DM260_PB_Result_Data_64_bytes_1[69];
	PlcInputs.ST70_3_DM260_PB_Result_Data_64_bytes_1[70] := HwInputs.ST70_3_DM260_PB_Result_Data_64_bytes_1[70];
	PlcInputs.ST70_3_DM260_PB_Result_Data_64_bytes_1[71] := HwInputs.ST70_3_DM260_PB_Result_Data_64_bytes_1[71];
	PlcInputs.ST70_1_DM260_EB_Acquisition_Status_1[0] := HwInputs.ST70_1_DM260_EB_Acquisition_Status_1[0];
	PlcInputs.ST70_1_DM260_EB_Acquisition_Status_1[1] := HwInputs.ST70_1_DM260_EB_Acquisition_Status_1[1];
	PlcInputs.ST70_1_DM260_EB_Acquisition_Status_1[2] := HwInputs.ST70_1_DM260_EB_Acquisition_Status_1[2];
	PlcInputs.ST70_1_DM260_EB_Results_Status_1 := HwInputs.ST70_1_DM260_EB_Results_Status_1;
	PlcInputs.ST70_1_DM260_EB_Soft_Event_Control_1 := HwInputs.ST70_1_DM260_EB_Soft_Event_Control_1;
	PlcInputs.ST70_1_DM260_EB_Result_Data_64_bytes_1[0] := HwInputs.ST70_1_DM260_EB_Result_Data_64_bytes_1[0];
	PlcInputs.ST70_1_DM260_EB_Result_Data_64_bytes_1[1] := HwInputs.ST70_1_DM260_EB_Result_Data_64_bytes_1[1];
	PlcInputs.ST70_1_DM260_EB_Result_Data_64_bytes_1[2] := HwInputs.ST70_1_DM260_EB_Result_Data_64_bytes_1[2];
	PlcInputs.ST70_1_DM260_EB_Result_Data_64_bytes_1[3] := HwInputs.ST70_1_DM260_EB_Result_Data_64_bytes_1[3];
	PlcInputs.ST70_1_DM260_EB_Result_Data_64_bytes_1[4] := HwInputs.ST70_1_DM260_EB_Result_Data_64_bytes_1[4];
	PlcInputs.ST70_1_DM260_EB_Result_Data_64_bytes_1[5] := HwInputs.ST70_1_DM260_EB_Result_Data_64_bytes_1[5];
	PlcInputs.ST70_1_DM260_EB_Result_Data_64_bytes_1[6] := HwInputs.ST70_1_DM260_EB_Result_Data_64_bytes_1[6];
	PlcInputs.ST70_1_DM260_EB_Result_Data_64_bytes_1[7] := HwInputs.ST70_1_DM260_EB_Result_Data_64_bytes_1[7];
	PlcInputs.ST70_1_DM260_EB_Result_Data_64_bytes_1[8] := HwInputs.ST70_1_DM260_EB_Result_Data_64_bytes_1[8];
	PlcInputs.ST70_1_DM260_EB_Result_Data_64_bytes_1[9] := HwInputs.ST70_1_DM260_EB_Result_Data_64_bytes_1[9];
	PlcInputs.ST70_1_DM260_EB_Result_Data_64_bytes_1[10] := HwInputs.ST70_1_DM260_EB_Result_Data_64_bytes_1[10];
	PlcInputs.ST70_1_DM260_EB_Result_Data_64_bytes_1[11] := HwInputs.ST70_1_DM260_EB_Result_Data_64_bytes_1[11];
	PlcInputs.ST70_1_DM260_EB_Result_Data_64_bytes_1[12] := HwInputs.ST70_1_DM260_EB_Result_Data_64_bytes_1[12];
	PlcInputs.ST70_1_DM260_EB_Result_Data_64_bytes_1[13] := HwInputs.ST70_1_DM260_EB_Result_Data_64_bytes_1[13];
	PlcInputs.ST70_1_DM260_EB_Result_Data_64_bytes_1[14] := HwInputs.ST70_1_DM260_EB_Result_Data_64_bytes_1[14];
	PlcInputs.ST70_1_DM260_EB_Result_Data_64_bytes_1[15] := HwInputs.ST70_1_DM260_EB_Result_Data_64_bytes_1[15];
	PlcInputs.ST70_1_DM260_EB_Result_Data_64_bytes_1[16] := HwInputs.ST70_1_DM260_EB_Result_Data_64_bytes_1[16];
	PlcInputs.ST70_1_DM260_EB_Result_Data_64_bytes_1[17] := HwInputs.ST70_1_DM260_EB_Result_Data_64_bytes_1[17];
	PlcInputs.ST70_1_DM260_EB_Result_Data_64_bytes_1[18] := HwInputs.ST70_1_DM260_EB_Result_Data_64_bytes_1[18];
	PlcInputs.ST70_1_DM260_EB_Result_Data_64_bytes_1[19] := HwInputs.ST70_1_DM260_EB_Result_Data_64_bytes_1[19];
	PlcInputs.ST70_1_DM260_EB_Result_Data_64_bytes_1[20] := HwInputs.ST70_1_DM260_EB_Result_Data_64_bytes_1[20];
	PlcInputs.ST70_1_DM260_EB_Result_Data_64_bytes_1[21] := HwInputs.ST70_1_DM260_EB_Result_Data_64_bytes_1[21];
	PlcInputs.ST70_1_DM260_EB_Result_Data_64_bytes_1[22] := HwInputs.ST70_1_DM260_EB_Result_Data_64_bytes_1[22];
	PlcInputs.ST70_1_DM260_EB_Result_Data_64_bytes_1[23] := HwInputs.ST70_1_DM260_EB_Result_Data_64_bytes_1[23];
	PlcInputs.ST70_1_DM260_EB_Result_Data_64_bytes_1[24] := HwInputs.ST70_1_DM260_EB_Result_Data_64_bytes_1[24];
	PlcInputs.ST70_1_DM260_EB_Result_Data_64_bytes_1[25] := HwInputs.ST70_1_DM260_EB_Result_Data_64_bytes_1[25];
	PlcInputs.ST70_1_DM260_EB_Result_Data_64_bytes_1[26] := HwInputs.ST70_1_DM260_EB_Result_Data_64_bytes_1[26];
	PlcInputs.ST70_1_DM260_EB_Result_Data_64_bytes_1[27] := HwInputs.ST70_1_DM260_EB_Result_Data_64_bytes_1[27];
	PlcInputs.ST70_1_DM260_EB_Result_Data_64_bytes_1[28] := HwInputs.ST70_1_DM260_EB_Result_Data_64_bytes_1[28];
	PlcInputs.ST70_1_DM260_EB_Result_Data_64_bytes_1[29] := HwInputs.ST70_1_DM260_EB_Result_Data_64_bytes_1[29];
	PlcInputs.ST70_1_DM260_EB_Result_Data_64_bytes_1[30] := HwInputs.ST70_1_DM260_EB_Result_Data_64_bytes_1[30];
	PlcInputs.ST70_1_DM260_EB_Result_Data_64_bytes_1[31] := HwInputs.ST70_1_DM260_EB_Result_Data_64_bytes_1[31];
	PlcInputs.ST70_1_DM260_EB_Result_Data_64_bytes_1[32] := HwInputs.ST70_1_DM260_EB_Result_Data_64_bytes_1[32];
	PlcInputs.ST70_1_DM260_EB_Result_Data_64_bytes_1[33] := HwInputs.ST70_1_DM260_EB_Result_Data_64_bytes_1[33];
	PlcInputs.ST70_1_DM260_EB_Result_Data_64_bytes_1[34] := HwInputs.ST70_1_DM260_EB_Result_Data_64_bytes_1[34];
	PlcInputs.ST70_1_DM260_EB_Result_Data_64_bytes_1[35] := HwInputs.ST70_1_DM260_EB_Result_Data_64_bytes_1[35];
	PlcInputs.ST70_1_DM260_EB_Result_Data_64_bytes_1[36] := HwInputs.ST70_1_DM260_EB_Result_Data_64_bytes_1[36];
	PlcInputs.ST70_1_DM260_EB_Result_Data_64_bytes_1[37] := HwInputs.ST70_1_DM260_EB_Result_Data_64_bytes_1[37];
	PlcInputs.ST70_1_DM260_EB_Result_Data_64_bytes_1[38] := HwInputs.ST70_1_DM260_EB_Result_Data_64_bytes_1[38];
	PlcInputs.ST70_1_DM260_EB_Result_Data_64_bytes_1[39] := HwInputs.ST70_1_DM260_EB_Result_Data_64_bytes_1[39];
	PlcInputs.ST70_1_DM260_EB_Result_Data_64_bytes_1[40] := HwInputs.ST70_1_DM260_EB_Result_Data_64_bytes_1[40];
	PlcInputs.ST70_1_DM260_EB_Result_Data_64_bytes_1[41] := HwInputs.ST70_1_DM260_EB_Result_Data_64_bytes_1[41];
	PlcInputs.ST70_1_DM260_EB_Result_Data_64_bytes_1[42] := HwInputs.ST70_1_DM260_EB_Result_Data_64_bytes_1[42];
	PlcInputs.ST70_1_DM260_EB_Result_Data_64_bytes_1[43] := HwInputs.ST70_1_DM260_EB_Result_Data_64_bytes_1[43];
	PlcInputs.ST70_1_DM260_EB_Result_Data_64_bytes_1[44] := HwInputs.ST70_1_DM260_EB_Result_Data_64_bytes_1[44];
	PlcInputs.ST70_1_DM260_EB_Result_Data_64_bytes_1[45] := HwInputs.ST70_1_DM260_EB_Result_Data_64_bytes_1[45];
	PlcInputs.ST70_1_DM260_EB_Result_Data_64_bytes_1[46] := HwInputs.ST70_1_DM260_EB_Result_Data_64_bytes_1[46];
	PlcInputs.ST70_1_DM260_EB_Result_Data_64_bytes_1[47] := HwInputs.ST70_1_DM260_EB_Result_Data_64_bytes_1[47];
	PlcInputs.ST70_1_DM260_EB_Result_Data_64_bytes_1[48] := HwInputs.ST70_1_DM260_EB_Result_Data_64_bytes_1[48];
	PlcInputs.ST70_1_DM260_EB_Result_Data_64_bytes_1[49] := HwInputs.ST70_1_DM260_EB_Result_Data_64_bytes_1[49];
	PlcInputs.ST70_1_DM260_EB_Result_Data_64_bytes_1[50] := HwInputs.ST70_1_DM260_EB_Result_Data_64_bytes_1[50];
	PlcInputs.ST70_1_DM260_EB_Result_Data_64_bytes_1[51] := HwInputs.ST70_1_DM260_EB_Result_Data_64_bytes_1[51];
	PlcInputs.ST70_1_DM260_EB_Result_Data_64_bytes_1[52] := HwInputs.ST70_1_DM260_EB_Result_Data_64_bytes_1[52];
	PlcInputs.ST70_1_DM260_EB_Result_Data_64_bytes_1[53] := HwInputs.ST70_1_DM260_EB_Result_Data_64_bytes_1[53];
	PlcInputs.ST70_1_DM260_EB_Result_Data_64_bytes_1[54] := HwInputs.ST70_1_DM260_EB_Result_Data_64_bytes_1[54];
	PlcInputs.ST70_1_DM260_EB_Result_Data_64_bytes_1[55] := HwInputs.ST70_1_DM260_EB_Result_Data_64_bytes_1[55];
	PlcInputs.ST70_1_DM260_EB_Result_Data_64_bytes_1[56] := HwInputs.ST70_1_DM260_EB_Result_Data_64_bytes_1[56];
	PlcInputs.ST70_1_DM260_EB_Result_Data_64_bytes_1[57] := HwInputs.ST70_1_DM260_EB_Result_Data_64_bytes_1[57];
	PlcInputs.ST70_1_DM260_EB_Result_Data_64_bytes_1[58] := HwInputs.ST70_1_DM260_EB_Result_Data_64_bytes_1[58];
	PlcInputs.ST70_1_DM260_EB_Result_Data_64_bytes_1[59] := HwInputs.ST70_1_DM260_EB_Result_Data_64_bytes_1[59];
	PlcInputs.ST70_1_DM260_EB_Result_Data_64_bytes_1[60] := HwInputs.ST70_1_DM260_EB_Result_Data_64_bytes_1[60];
	PlcInputs.ST70_1_DM260_EB_Result_Data_64_bytes_1[61] := HwInputs.ST70_1_DM260_EB_Result_Data_64_bytes_1[61];
	PlcInputs.ST70_1_DM260_EB_Result_Data_64_bytes_1[62] := HwInputs.ST70_1_DM260_EB_Result_Data_64_bytes_1[62];
	PlcInputs.ST70_1_DM260_EB_Result_Data_64_bytes_1[63] := HwInputs.ST70_1_DM260_EB_Result_Data_64_bytes_1[63];
	PlcInputs.ST70_1_DM260_EB_Result_Data_64_bytes_1[64] := HwInputs.ST70_1_DM260_EB_Result_Data_64_bytes_1[64];
	PlcInputs.ST70_1_DM260_EB_Result_Data_64_bytes_1[65] := HwInputs.ST70_1_DM260_EB_Result_Data_64_bytes_1[65];
	PlcInputs.ST70_1_DM260_EB_Result_Data_64_bytes_1[66] := HwInputs.ST70_1_DM260_EB_Result_Data_64_bytes_1[66];
	PlcInputs.ST70_1_DM260_EB_Result_Data_64_bytes_1[67] := HwInputs.ST70_1_DM260_EB_Result_Data_64_bytes_1[67];
	PlcInputs.ST70_1_DM260_EB_Result_Data_64_bytes_1[68] := HwInputs.ST70_1_DM260_EB_Result_Data_64_bytes_1[68];
	PlcInputs.ST70_1_DM260_EB_Result_Data_64_bytes_1[69] := HwInputs.ST70_1_DM260_EB_Result_Data_64_bytes_1[69];
	PlcInputs.ST70_1_DM260_EB_Result_Data_64_bytes_1[70] := HwInputs.ST70_1_DM260_EB_Result_Data_64_bytes_1[70];
	PlcInputs.ST70_1_DM260_EB_Result_Data_64_bytes_1[71] := HwInputs.ST70_1_DM260_EB_Result_Data_64_bytes_1[71];
	PlcInputs.ST70_2_DM260_EB_Acquisition_Status_1[0] := HwInputs.ST70_2_DM260_EB_Acquisition_Status_1[0];
	PlcInputs.ST70_2_DM260_EB_Acquisition_Status_1[1] := HwInputs.ST70_2_DM260_EB_Acquisition_Status_1[1];
	PlcInputs.ST70_2_DM260_EB_Acquisition_Status_1[2] := HwInputs.ST70_2_DM260_EB_Acquisition_Status_1[2];
	PlcInputs.ST70_2_DM260_EB_Results_Status_1 := HwInputs.ST70_2_DM260_EB_Results_Status_1;
	PlcInputs.ST70_2_DM260_EB_Soft_Event_Control_1 := HwInputs.ST70_2_DM260_EB_Soft_Event_Control_1;
	PlcInputs.ST70_2_DM260_EB_Result_Data_64_bytes_1[0] := HwInputs.ST70_2_DM260_EB_Result_Data_64_bytes_1[0];
	PlcInputs.ST70_2_DM260_EB_Result_Data_64_bytes_1[1] := HwInputs.ST70_2_DM260_EB_Result_Data_64_bytes_1[1];
	PlcInputs.ST70_2_DM260_EB_Result_Data_64_bytes_1[2] := HwInputs.ST70_2_DM260_EB_Result_Data_64_bytes_1[2];
	PlcInputs.ST70_2_DM260_EB_Result_Data_64_bytes_1[3] := HwInputs.ST70_2_DM260_EB_Result_Data_64_bytes_1[3];
	PlcInputs.ST70_2_DM260_EB_Result_Data_64_bytes_1[4] := HwInputs.ST70_2_DM260_EB_Result_Data_64_bytes_1[4];
	PlcInputs.ST70_2_DM260_EB_Result_Data_64_bytes_1[5] := HwInputs.ST70_2_DM260_EB_Result_Data_64_bytes_1[5];
	PlcInputs.ST70_2_DM260_EB_Result_Data_64_bytes_1[6] := HwInputs.ST70_2_DM260_EB_Result_Data_64_bytes_1[6];
	PlcInputs.ST70_2_DM260_EB_Result_Data_64_bytes_1[7] := HwInputs.ST70_2_DM260_EB_Result_Data_64_bytes_1[7];
	PlcInputs.ST70_2_DM260_EB_Result_Data_64_bytes_1[8] := HwInputs.ST70_2_DM260_EB_Result_Data_64_bytes_1[8];
	PlcInputs.ST70_2_DM260_EB_Result_Data_64_bytes_1[9] := HwInputs.ST70_2_DM260_EB_Result_Data_64_bytes_1[9];
	PlcInputs.ST70_2_DM260_EB_Result_Data_64_bytes_1[10] := HwInputs.ST70_2_DM260_EB_Result_Data_64_bytes_1[10];
	PlcInputs.ST70_2_DM260_EB_Result_Data_64_bytes_1[11] := HwInputs.ST70_2_DM260_EB_Result_Data_64_bytes_1[11];
	PlcInputs.ST70_2_DM260_EB_Result_Data_64_bytes_1[12] := HwInputs.ST70_2_DM260_EB_Result_Data_64_bytes_1[12];
	PlcInputs.ST70_2_DM260_EB_Result_Data_64_bytes_1[13] := HwInputs.ST70_2_DM260_EB_Result_Data_64_bytes_1[13];
	PlcInputs.ST70_2_DM260_EB_Result_Data_64_bytes_1[14] := HwInputs.ST70_2_DM260_EB_Result_Data_64_bytes_1[14];
	PlcInputs.ST70_2_DM260_EB_Result_Data_64_bytes_1[15] := HwInputs.ST70_2_DM260_EB_Result_Data_64_bytes_1[15];
	PlcInputs.ST70_2_DM260_EB_Result_Data_64_bytes_1[16] := HwInputs.ST70_2_DM260_EB_Result_Data_64_bytes_1[16];
	PlcInputs.ST70_2_DM260_EB_Result_Data_64_bytes_1[17] := HwInputs.ST70_2_DM260_EB_Result_Data_64_bytes_1[17];
	PlcInputs.ST70_2_DM260_EB_Result_Data_64_bytes_1[18] := HwInputs.ST70_2_DM260_EB_Result_Data_64_bytes_1[18];
	PlcInputs.ST70_2_DM260_EB_Result_Data_64_bytes_1[19] := HwInputs.ST70_2_DM260_EB_Result_Data_64_bytes_1[19];
	PlcInputs.ST70_2_DM260_EB_Result_Data_64_bytes_1[20] := HwInputs.ST70_2_DM260_EB_Result_Data_64_bytes_1[20];
	PlcInputs.ST70_2_DM260_EB_Result_Data_64_bytes_1[21] := HwInputs.ST70_2_DM260_EB_Result_Data_64_bytes_1[21];
	PlcInputs.ST70_2_DM260_EB_Result_Data_64_bytes_1[22] := HwInputs.ST70_2_DM260_EB_Result_Data_64_bytes_1[22];
	PlcInputs.ST70_2_DM260_EB_Result_Data_64_bytes_1[23] := HwInputs.ST70_2_DM260_EB_Result_Data_64_bytes_1[23];
	PlcInputs.ST70_2_DM260_EB_Result_Data_64_bytes_1[24] := HwInputs.ST70_2_DM260_EB_Result_Data_64_bytes_1[24];
	PlcInputs.ST70_2_DM260_EB_Result_Data_64_bytes_1[25] := HwInputs.ST70_2_DM260_EB_Result_Data_64_bytes_1[25];
	PlcInputs.ST70_2_DM260_EB_Result_Data_64_bytes_1[26] := HwInputs.ST70_2_DM260_EB_Result_Data_64_bytes_1[26];
	PlcInputs.ST70_2_DM260_EB_Result_Data_64_bytes_1[27] := HwInputs.ST70_2_DM260_EB_Result_Data_64_bytes_1[27];
	PlcInputs.ST70_2_DM260_EB_Result_Data_64_bytes_1[28] := HwInputs.ST70_2_DM260_EB_Result_Data_64_bytes_1[28];
	PlcInputs.ST70_2_DM260_EB_Result_Data_64_bytes_1[29] := HwInputs.ST70_2_DM260_EB_Result_Data_64_bytes_1[29];
	PlcInputs.ST70_2_DM260_EB_Result_Data_64_bytes_1[30] := HwInputs.ST70_2_DM260_EB_Result_Data_64_bytes_1[30];
	PlcInputs.ST70_2_DM260_EB_Result_Data_64_bytes_1[31] := HwInputs.ST70_2_DM260_EB_Result_Data_64_bytes_1[31];
	PlcInputs.ST70_2_DM260_EB_Result_Data_64_bytes_1[32] := HwInputs.ST70_2_DM260_EB_Result_Data_64_bytes_1[32];
	PlcInputs.ST70_2_DM260_EB_Result_Data_64_bytes_1[33] := HwInputs.ST70_2_DM260_EB_Result_Data_64_bytes_1[33];
	PlcInputs.ST70_2_DM260_EB_Result_Data_64_bytes_1[34] := HwInputs.ST70_2_DM260_EB_Result_Data_64_bytes_1[34];
	PlcInputs.ST70_2_DM260_EB_Result_Data_64_bytes_1[35] := HwInputs.ST70_2_DM260_EB_Result_Data_64_bytes_1[35];
	PlcInputs.ST70_2_DM260_EB_Result_Data_64_bytes_1[36] := HwInputs.ST70_2_DM260_EB_Result_Data_64_bytes_1[36];
	PlcInputs.ST70_2_DM260_EB_Result_Data_64_bytes_1[37] := HwInputs.ST70_2_DM260_EB_Result_Data_64_bytes_1[37];
	PlcInputs.ST70_2_DM260_EB_Result_Data_64_bytes_1[38] := HwInputs.ST70_2_DM260_EB_Result_Data_64_bytes_1[38];
	PlcInputs.ST70_2_DM260_EB_Result_Data_64_bytes_1[39] := HwInputs.ST70_2_DM260_EB_Result_Data_64_bytes_1[39];
	PlcInputs.ST70_2_DM260_EB_Result_Data_64_bytes_1[40] := HwInputs.ST70_2_DM260_EB_Result_Data_64_bytes_1[40];
	PlcInputs.ST70_2_DM260_EB_Result_Data_64_bytes_1[41] := HwInputs.ST70_2_DM260_EB_Result_Data_64_bytes_1[41];
	PlcInputs.ST70_2_DM260_EB_Result_Data_64_bytes_1[42] := HwInputs.ST70_2_DM260_EB_Result_Data_64_bytes_1[42];
	PlcInputs.ST70_2_DM260_EB_Result_Data_64_bytes_1[43] := HwInputs.ST70_2_DM260_EB_Result_Data_64_bytes_1[43];
	PlcInputs.ST70_2_DM260_EB_Result_Data_64_bytes_1[44] := HwInputs.ST70_2_DM260_EB_Result_Data_64_bytes_1[44];
	PlcInputs.ST70_2_DM260_EB_Result_Data_64_bytes_1[45] := HwInputs.ST70_2_DM260_EB_Result_Data_64_bytes_1[45];
	PlcInputs.ST70_2_DM260_EB_Result_Data_64_bytes_1[46] := HwInputs.ST70_2_DM260_EB_Result_Data_64_bytes_1[46];
	PlcInputs.ST70_2_DM260_EB_Result_Data_64_bytes_1[47] := HwInputs.ST70_2_DM260_EB_Result_Data_64_bytes_1[47];
	PlcInputs.ST70_2_DM260_EB_Result_Data_64_bytes_1[48] := HwInputs.ST70_2_DM260_EB_Result_Data_64_bytes_1[48];
	PlcInputs.ST70_2_DM260_EB_Result_Data_64_bytes_1[49] := HwInputs.ST70_2_DM260_EB_Result_Data_64_bytes_1[49];
	PlcInputs.ST70_2_DM260_EB_Result_Data_64_bytes_1[50] := HwInputs.ST70_2_DM260_EB_Result_Data_64_bytes_1[50];
	PlcInputs.ST70_2_DM260_EB_Result_Data_64_bytes_1[51] := HwInputs.ST70_2_DM260_EB_Result_Data_64_bytes_1[51];
	PlcInputs.ST70_2_DM260_EB_Result_Data_64_bytes_1[52] := HwInputs.ST70_2_DM260_EB_Result_Data_64_bytes_1[52];
	PlcInputs.ST70_2_DM260_EB_Result_Data_64_bytes_1[53] := HwInputs.ST70_2_DM260_EB_Result_Data_64_bytes_1[53];
	PlcInputs.ST70_2_DM260_EB_Result_Data_64_bytes_1[54] := HwInputs.ST70_2_DM260_EB_Result_Data_64_bytes_1[54];
	PlcInputs.ST70_2_DM260_EB_Result_Data_64_bytes_1[55] := HwInputs.ST70_2_DM260_EB_Result_Data_64_bytes_1[55];
	PlcInputs.ST70_2_DM260_EB_Result_Data_64_bytes_1[56] := HwInputs.ST70_2_DM260_EB_Result_Data_64_bytes_1[56];
	PlcInputs.ST70_2_DM260_EB_Result_Data_64_bytes_1[57] := HwInputs.ST70_2_DM260_EB_Result_Data_64_bytes_1[57];
	PlcInputs.ST70_2_DM260_EB_Result_Data_64_bytes_1[58] := HwInputs.ST70_2_DM260_EB_Result_Data_64_bytes_1[58];
	PlcInputs.ST70_2_DM260_EB_Result_Data_64_bytes_1[59] := HwInputs.ST70_2_DM260_EB_Result_Data_64_bytes_1[59];
	PlcInputs.ST70_2_DM260_EB_Result_Data_64_bytes_1[60] := HwInputs.ST70_2_DM260_EB_Result_Data_64_bytes_1[60];
	PlcInputs.ST70_2_DM260_EB_Result_Data_64_bytes_1[61] := HwInputs.ST70_2_DM260_EB_Result_Data_64_bytes_1[61];
	PlcInputs.ST70_2_DM260_EB_Result_Data_64_bytes_1[62] := HwInputs.ST70_2_DM260_EB_Result_Data_64_bytes_1[62];
	PlcInputs.ST70_2_DM260_EB_Result_Data_64_bytes_1[63] := HwInputs.ST70_2_DM260_EB_Result_Data_64_bytes_1[63];
	PlcInputs.ST70_2_DM260_EB_Result_Data_64_bytes_1[64] := HwInputs.ST70_2_DM260_EB_Result_Data_64_bytes_1[64];
	PlcInputs.ST70_2_DM260_EB_Result_Data_64_bytes_1[65] := HwInputs.ST70_2_DM260_EB_Result_Data_64_bytes_1[65];
	PlcInputs.ST70_2_DM260_EB_Result_Data_64_bytes_1[66] := HwInputs.ST70_2_DM260_EB_Result_Data_64_bytes_1[66];
	PlcInputs.ST70_2_DM260_EB_Result_Data_64_bytes_1[67] := HwInputs.ST70_2_DM260_EB_Result_Data_64_bytes_1[67];
	PlcInputs.ST70_2_DM260_EB_Result_Data_64_bytes_1[68] := HwInputs.ST70_2_DM260_EB_Result_Data_64_bytes_1[68];
	PlcInputs.ST70_2_DM260_EB_Result_Data_64_bytes_1[69] := HwInputs.ST70_2_DM260_EB_Result_Data_64_bytes_1[69];
	PlcInputs.ST70_2_DM260_EB_Result_Data_64_bytes_1[70] := HwInputs.ST70_2_DM260_EB_Result_Data_64_bytes_1[70];
	PlcInputs.ST70_2_DM260_EB_Result_Data_64_bytes_1[71] := HwInputs.ST70_2_DM260_EB_Result_Data_64_bytes_1[71];
	PlcInputs.ST70_3_DM260_EB_Acquisition_Status_1[0] := HwInputs.ST70_3_DM260_EB_Acquisition_Status_1[0];
	PlcInputs.ST70_3_DM260_EB_Acquisition_Status_1[1] := HwInputs.ST70_3_DM260_EB_Acquisition_Status_1[1];
	PlcInputs.ST70_3_DM260_EB_Acquisition_Status_1[2] := HwInputs.ST70_3_DM260_EB_Acquisition_Status_1[2];
	PlcInputs.ST70_3_DM260_EB_Results_Status_1 := HwInputs.ST70_3_DM260_EB_Results_Status_1;
	PlcInputs.ST70_3_DM260_EB_Soft_Event_Control_1 := HwInputs.ST70_3_DM260_EB_Soft_Event_Control_1;
	PlcInputs.ST70_3_DM260_EB_Result_Data_64_bytes_1[0] := HwInputs.ST70_3_DM260_EB_Result_Data_64_bytes_1[0];
	PlcInputs.ST70_3_DM260_EB_Result_Data_64_bytes_1[1] := HwInputs.ST70_3_DM260_EB_Result_Data_64_bytes_1[1];
	PlcInputs.ST70_3_DM260_EB_Result_Data_64_bytes_1[2] := HwInputs.ST70_3_DM260_EB_Result_Data_64_bytes_1[2];
	PlcInputs.ST70_3_DM260_EB_Result_Data_64_bytes_1[3] := HwInputs.ST70_3_DM260_EB_Result_Data_64_bytes_1[3];
	PlcInputs.ST70_3_DM260_EB_Result_Data_64_bytes_1[4] := HwInputs.ST70_3_DM260_EB_Result_Data_64_bytes_1[4];
	PlcInputs.ST70_3_DM260_EB_Result_Data_64_bytes_1[5] := HwInputs.ST70_3_DM260_EB_Result_Data_64_bytes_1[5];
	PlcInputs.ST70_3_DM260_EB_Result_Data_64_bytes_1[6] := HwInputs.ST70_3_DM260_EB_Result_Data_64_bytes_1[6];
	PlcInputs.ST70_3_DM260_EB_Result_Data_64_bytes_1[7] := HwInputs.ST70_3_DM260_EB_Result_Data_64_bytes_1[7];
	PlcInputs.ST70_3_DM260_EB_Result_Data_64_bytes_1[8] := HwInputs.ST70_3_DM260_EB_Result_Data_64_bytes_1[8];
	PlcInputs.ST70_3_DM260_EB_Result_Data_64_bytes_1[9] := HwInputs.ST70_3_DM260_EB_Result_Data_64_bytes_1[9];
	PlcInputs.ST70_3_DM260_EB_Result_Data_64_bytes_1[10] := HwInputs.ST70_3_DM260_EB_Result_Data_64_bytes_1[10];
	PlcInputs.ST70_3_DM260_EB_Result_Data_64_bytes_1[11] := HwInputs.ST70_3_DM260_EB_Result_Data_64_bytes_1[11];
	PlcInputs.ST70_3_DM260_EB_Result_Data_64_bytes_1[12] := HwInputs.ST70_3_DM260_EB_Result_Data_64_bytes_1[12];
	PlcInputs.ST70_3_DM260_EB_Result_Data_64_bytes_1[13] := HwInputs.ST70_3_DM260_EB_Result_Data_64_bytes_1[13];
	PlcInputs.ST70_3_DM260_EB_Result_Data_64_bytes_1[14] := HwInputs.ST70_3_DM260_EB_Result_Data_64_bytes_1[14];
	PlcInputs.ST70_3_DM260_EB_Result_Data_64_bytes_1[15] := HwInputs.ST70_3_DM260_EB_Result_Data_64_bytes_1[15];
	PlcInputs.ST70_3_DM260_EB_Result_Data_64_bytes_1[16] := HwInputs.ST70_3_DM260_EB_Result_Data_64_bytes_1[16];
	PlcInputs.ST70_3_DM260_EB_Result_Data_64_bytes_1[17] := HwInputs.ST70_3_DM260_EB_Result_Data_64_bytes_1[17];
	PlcInputs.ST70_3_DM260_EB_Result_Data_64_bytes_1[18] := HwInputs.ST70_3_DM260_EB_Result_Data_64_bytes_1[18];
	PlcInputs.ST70_3_DM260_EB_Result_Data_64_bytes_1[19] := HwInputs.ST70_3_DM260_EB_Result_Data_64_bytes_1[19];
	PlcInputs.ST70_3_DM260_EB_Result_Data_64_bytes_1[20] := HwInputs.ST70_3_DM260_EB_Result_Data_64_bytes_1[20];
	PlcInputs.ST70_3_DM260_EB_Result_Data_64_bytes_1[21] := HwInputs.ST70_3_DM260_EB_Result_Data_64_bytes_1[21];
	PlcInputs.ST70_3_DM260_EB_Result_Data_64_bytes_1[22] := HwInputs.ST70_3_DM260_EB_Result_Data_64_bytes_1[22];
	PlcInputs.ST70_3_DM260_EB_Result_Data_64_bytes_1[23] := HwInputs.ST70_3_DM260_EB_Result_Data_64_bytes_1[23];
	PlcInputs.ST70_3_DM260_EB_Result_Data_64_bytes_1[24] := HwInputs.ST70_3_DM260_EB_Result_Data_64_bytes_1[24];
	PlcInputs.ST70_3_DM260_EB_Result_Data_64_bytes_1[25] := HwInputs.ST70_3_DM260_EB_Result_Data_64_bytes_1[25];
	PlcInputs.ST70_3_DM260_EB_Result_Data_64_bytes_1[26] := HwInputs.ST70_3_DM260_EB_Result_Data_64_bytes_1[26];
	PlcInputs.ST70_3_DM260_EB_Result_Data_64_bytes_1[27] := HwInputs.ST70_3_DM260_EB_Result_Data_64_bytes_1[27];
	PlcInputs.ST70_3_DM260_EB_Result_Data_64_bytes_1[28] := HwInputs.ST70_3_DM260_EB_Result_Data_64_bytes_1[28];
	PlcInputs.ST70_3_DM260_EB_Result_Data_64_bytes_1[29] := HwInputs.ST70_3_DM260_EB_Result_Data_64_bytes_1[29];
	PlcInputs.ST70_3_DM260_EB_Result_Data_64_bytes_1[30] := HwInputs.ST70_3_DM260_EB_Result_Data_64_bytes_1[30];
	PlcInputs.ST70_3_DM260_EB_Result_Data_64_bytes_1[31] := HwInputs.ST70_3_DM260_EB_Result_Data_64_bytes_1[31];
	PlcInputs.ST70_3_DM260_EB_Result_Data_64_bytes_1[32] := HwInputs.ST70_3_DM260_EB_Result_Data_64_bytes_1[32];
	PlcInputs.ST70_3_DM260_EB_Result_Data_64_bytes_1[33] := HwInputs.ST70_3_DM260_EB_Result_Data_64_bytes_1[33];
	PlcInputs.ST70_3_DM260_EB_Result_Data_64_bytes_1[34] := HwInputs.ST70_3_DM260_EB_Result_Data_64_bytes_1[34];
	PlcInputs.ST70_3_DM260_EB_Result_Data_64_bytes_1[35] := HwInputs.ST70_3_DM260_EB_Result_Data_64_bytes_1[35];
	PlcInputs.ST70_3_DM260_EB_Result_Data_64_bytes_1[36] := HwInputs.ST70_3_DM260_EB_Result_Data_64_bytes_1[36];
	PlcInputs.ST70_3_DM260_EB_Result_Data_64_bytes_1[37] := HwInputs.ST70_3_DM260_EB_Result_Data_64_bytes_1[37];
	PlcInputs.ST70_3_DM260_EB_Result_Data_64_bytes_1[38] := HwInputs.ST70_3_DM260_EB_Result_Data_64_bytes_1[38];
	PlcInputs.ST70_3_DM260_EB_Result_Data_64_bytes_1[39] := HwInputs.ST70_3_DM260_EB_Result_Data_64_bytes_1[39];
	PlcInputs.ST70_3_DM260_EB_Result_Data_64_bytes_1[40] := HwInputs.ST70_3_DM260_EB_Result_Data_64_bytes_1[40];
	PlcInputs.ST70_3_DM260_EB_Result_Data_64_bytes_1[41] := HwInputs.ST70_3_DM260_EB_Result_Data_64_bytes_1[41];
	PlcInputs.ST70_3_DM260_EB_Result_Data_64_bytes_1[42] := HwInputs.ST70_3_DM260_EB_Result_Data_64_bytes_1[42];
	PlcInputs.ST70_3_DM260_EB_Result_Data_64_bytes_1[43] := HwInputs.ST70_3_DM260_EB_Result_Data_64_bytes_1[43];
	PlcInputs.ST70_3_DM260_EB_Result_Data_64_bytes_1[44] := HwInputs.ST70_3_DM260_EB_Result_Data_64_bytes_1[44];
	PlcInputs.ST70_3_DM260_EB_Result_Data_64_bytes_1[45] := HwInputs.ST70_3_DM260_EB_Result_Data_64_bytes_1[45];
	PlcInputs.ST70_3_DM260_EB_Result_Data_64_bytes_1[46] := HwInputs.ST70_3_DM260_EB_Result_Data_64_bytes_1[46];
	PlcInputs.ST70_3_DM260_EB_Result_Data_64_bytes_1[47] := HwInputs.ST70_3_DM260_EB_Result_Data_64_bytes_1[47];
	PlcInputs.ST70_3_DM260_EB_Result_Data_64_bytes_1[48] := HwInputs.ST70_3_DM260_EB_Result_Data_64_bytes_1[48];
	PlcInputs.ST70_3_DM260_EB_Result_Data_64_bytes_1[49] := HwInputs.ST70_3_DM260_EB_Result_Data_64_bytes_1[49];
	PlcInputs.ST70_3_DM260_EB_Result_Data_64_bytes_1[50] := HwInputs.ST70_3_DM260_EB_Result_Data_64_bytes_1[50];
	PlcInputs.ST70_3_DM260_EB_Result_Data_64_bytes_1[51] := HwInputs.ST70_3_DM260_EB_Result_Data_64_bytes_1[51];
	PlcInputs.ST70_3_DM260_EB_Result_Data_64_bytes_1[52] := HwInputs.ST70_3_DM260_EB_Result_Data_64_bytes_1[52];
	PlcInputs.ST70_3_DM260_EB_Result_Data_64_bytes_1[53] := HwInputs.ST70_3_DM260_EB_Result_Data_64_bytes_1[53];
	PlcInputs.ST70_3_DM260_EB_Result_Data_64_bytes_1[54] := HwInputs.ST70_3_DM260_EB_Result_Data_64_bytes_1[54];
	PlcInputs.ST70_3_DM260_EB_Result_Data_64_bytes_1[55] := HwInputs.ST70_3_DM260_EB_Result_Data_64_bytes_1[55];
	PlcInputs.ST70_3_DM260_EB_Result_Data_64_bytes_1[56] := HwInputs.ST70_3_DM260_EB_Result_Data_64_bytes_1[56];
	PlcInputs.ST70_3_DM260_EB_Result_Data_64_bytes_1[57] := HwInputs.ST70_3_DM260_EB_Result_Data_64_bytes_1[57];
	PlcInputs.ST70_3_DM260_EB_Result_Data_64_bytes_1[58] := HwInputs.ST70_3_DM260_EB_Result_Data_64_bytes_1[58];
	PlcInputs.ST70_3_DM260_EB_Result_Data_64_bytes_1[59] := HwInputs.ST70_3_DM260_EB_Result_Data_64_bytes_1[59];
	PlcInputs.ST70_3_DM260_EB_Result_Data_64_bytes_1[60] := HwInputs.ST70_3_DM260_EB_Result_Data_64_bytes_1[60];
	PlcInputs.ST70_3_DM260_EB_Result_Data_64_bytes_1[61] := HwInputs.ST70_3_DM260_EB_Result_Data_64_bytes_1[61];
	PlcInputs.ST70_3_DM260_EB_Result_Data_64_bytes_1[62] := HwInputs.ST70_3_DM260_EB_Result_Data_64_bytes_1[62];
	PlcInputs.ST70_3_DM260_EB_Result_Data_64_bytes_1[63] := HwInputs.ST70_3_DM260_EB_Result_Data_64_bytes_1[63];
	PlcInputs.ST70_3_DM260_EB_Result_Data_64_bytes_1[64] := HwInputs.ST70_3_DM260_EB_Result_Data_64_bytes_1[64];
	PlcInputs.ST70_3_DM260_EB_Result_Data_64_bytes_1[65] := HwInputs.ST70_3_DM260_EB_Result_Data_64_bytes_1[65];
	PlcInputs.ST70_3_DM260_EB_Result_Data_64_bytes_1[66] := HwInputs.ST70_3_DM260_EB_Result_Data_64_bytes_1[66];
	PlcInputs.ST70_3_DM260_EB_Result_Data_64_bytes_1[67] := HwInputs.ST70_3_DM260_EB_Result_Data_64_bytes_1[67];
	PlcInputs.ST70_3_DM260_EB_Result_Data_64_bytes_1[68] := HwInputs.ST70_3_DM260_EB_Result_Data_64_bytes_1[68];
	PlcInputs.ST70_3_DM260_EB_Result_Data_64_bytes_1[69] := HwInputs.ST70_3_DM260_EB_Result_Data_64_bytes_1[69];
	PlcInputs.ST70_3_DM260_EB_Result_Data_64_bytes_1[70] := HwInputs.ST70_3_DM260_EB_Result_Data_64_bytes_1[70];
	PlcInputs.ST70_3_DM260_EB_Result_Data_64_bytes_1[71] := HwInputs.ST70_3_DM260_EB_Result_Data_64_bytes_1[71];
	PlcInputs.ST70_1_CMMT_3GF3_DO_SERVO_1_Siemens_telegram_111_PZD_12_12[0] := HwInputs.ST70_1_CMMT_3GF3_DO_SERVO_1_Siemens_telegram_111_PZD_12_12[0];
	PlcInputs.ST70_1_CMMT_3GF3_DO_SERVO_1_Siemens_telegram_111_PZD_12_12[1] := HwInputs.ST70_1_CMMT_3GF3_DO_SERVO_1_Siemens_telegram_111_PZD_12_12[1];
	PlcInputs.ST70_1_CMMT_3GF3_DO_SERVO_1_Siemens_telegram_111_PZD_12_12[2] := HwInputs.ST70_1_CMMT_3GF3_DO_SERVO_1_Siemens_telegram_111_PZD_12_12[2];
	PlcInputs.ST70_1_CMMT_3GF3_DO_SERVO_1_Siemens_telegram_111_PZD_12_12[3] := HwInputs.ST70_1_CMMT_3GF3_DO_SERVO_1_Siemens_telegram_111_PZD_12_12[3];
	PlcInputs.ST70_1_CMMT_3GF3_DO_SERVO_1_Siemens_telegram_111_PZD_12_12[4] := HwInputs.ST70_1_CMMT_3GF3_DO_SERVO_1_Siemens_telegram_111_PZD_12_12[4];
	PlcInputs.ST70_1_CMMT_3GF3_DO_SERVO_1_Siemens_telegram_111_PZD_12_12[5] := HwInputs.ST70_1_CMMT_3GF3_DO_SERVO_1_Siemens_telegram_111_PZD_12_12[5];
	PlcInputs.ST70_1_CMMT_3GF3_DO_SERVO_1_Siemens_telegram_111_PZD_12_12[6] := HwInputs.ST70_1_CMMT_3GF3_DO_SERVO_1_Siemens_telegram_111_PZD_12_12[6];
	PlcInputs.ST70_1_CMMT_3GF3_DO_SERVO_1_Siemens_telegram_111_PZD_12_12[7] := HwInputs.ST70_1_CMMT_3GF3_DO_SERVO_1_Siemens_telegram_111_PZD_12_12[7];
	PlcInputs.ST70_1_CMMT_3GF3_DO_SERVO_1_Siemens_telegram_111_PZD_12_12[8] := HwInputs.ST70_1_CMMT_3GF3_DO_SERVO_1_Siemens_telegram_111_PZD_12_12[8];
	PlcInputs.ST70_1_CMMT_3GF3_DO_SERVO_1_Siemens_telegram_111_PZD_12_12[9] := HwInputs.ST70_1_CMMT_3GF3_DO_SERVO_1_Siemens_telegram_111_PZD_12_12[9];
	PlcInputs.ST70_1_CMMT_3GF3_DO_SERVO_1_Siemens_telegram_111_PZD_12_12[10] := HwInputs.ST70_1_CMMT_3GF3_DO_SERVO_1_Siemens_telegram_111_PZD_12_12[10];
	PlcInputs.ST70_1_CMMT_3GF3_DO_SERVO_1_Siemens_telegram_111_PZD_12_12[11] := HwInputs.ST70_1_CMMT_3GF3_DO_SERVO_1_Siemens_telegram_111_PZD_12_12[11];
	PlcInputs.ST70_1_CMMT_3GF3_DO_SERVO_1_Siemens_telegram_111_PZD_12_12[12] := HwInputs.ST70_1_CMMT_3GF3_DO_SERVO_1_Siemens_telegram_111_PZD_12_12[12];
	PlcInputs.ST70_1_CMMT_3GF3_DO_SERVO_1_Siemens_telegram_111_PZD_12_12[13] := HwInputs.ST70_1_CMMT_3GF3_DO_SERVO_1_Siemens_telegram_111_PZD_12_12[13];
	PlcInputs.ST70_1_CMMT_3GF3_DO_SERVO_1_Siemens_telegram_111_PZD_12_12[14] := HwInputs.ST70_1_CMMT_3GF3_DO_SERVO_1_Siemens_telegram_111_PZD_12_12[14];
	PlcInputs.ST70_1_CMMT_3GF3_DO_SERVO_1_Siemens_telegram_111_PZD_12_12[15] := HwInputs.ST70_1_CMMT_3GF3_DO_SERVO_1_Siemens_telegram_111_PZD_12_12[15];
	PlcInputs.ST70_1_CMMT_3GF3_DO_SERVO_1_Siemens_telegram_111_PZD_12_12[16] := HwInputs.ST70_1_CMMT_3GF3_DO_SERVO_1_Siemens_telegram_111_PZD_12_12[16];
	PlcInputs.ST70_1_CMMT_3GF3_DO_SERVO_1_Siemens_telegram_111_PZD_12_12[17] := HwInputs.ST70_1_CMMT_3GF3_DO_SERVO_1_Siemens_telegram_111_PZD_12_12[17];
	PlcInputs.ST70_1_CMMT_3GF3_DO_SERVO_1_Siemens_telegram_111_PZD_12_12[18] := HwInputs.ST70_1_CMMT_3GF3_DO_SERVO_1_Siemens_telegram_111_PZD_12_12[18];
	PlcInputs.ST70_1_CMMT_3GF3_DO_SERVO_1_Siemens_telegram_111_PZD_12_12[19] := HwInputs.ST70_1_CMMT_3GF3_DO_SERVO_1_Siemens_telegram_111_PZD_12_12[19];
	PlcInputs.ST70_1_CMMT_3GF3_DO_SERVO_1_Siemens_telegram_111_PZD_12_12[20] := HwInputs.ST70_1_CMMT_3GF3_DO_SERVO_1_Siemens_telegram_111_PZD_12_12[20];
	PlcInputs.ST70_1_CMMT_3GF3_DO_SERVO_1_Siemens_telegram_111_PZD_12_12[21] := HwInputs.ST70_1_CMMT_3GF3_DO_SERVO_1_Siemens_telegram_111_PZD_12_12[21];
	PlcInputs.ST70_1_CMMT_3GF3_DO_SERVO_1_Siemens_telegram_111_PZD_12_12[22] := HwInputs.ST70_1_CMMT_3GF3_DO_SERVO_1_Siemens_telegram_111_PZD_12_12[22];
	PlcInputs.ST70_1_CMMT_3GF3_DO_SERVO_1_Siemens_telegram_111_PZD_12_12[23] := HwInputs.ST70_1_CMMT_3GF3_DO_SERVO_1_Siemens_telegram_111_PZD_12_12[23];
END_FUNCTION
